FUNCTION_BLOCK "Controle_Dosagem_Complementos"   // FB7, FBD
{ S7_Optimized_Access := 'TRUE' }
VERSION : 0.1
   VAR_INPUT
      inEnable : Bool;
      inBotao_Externo : Bool;
      inValor_Atual_Balanca : Real;
   END_VAR
   VAR_OUTPUT
      outLedBotao_Externo : Bool;
   END_VAR
   VAR_IN_OUT
      Controle : Struct
         Quantidade_Itens : Int;   // Quantidade de complementos na receita
         Item_Atual : Int;   // Em qual item da receita esta no momento
         Quantidade_Dosada_Item_Atual : Real;   // Quantidade dosada do item atual, valor disponível após finalizado dosagem
         Habilitado_Inicio_Dosagem : Bool;   // Habilita o inicio da dosagem manual
         Botao_Inicio_Fim_Dosagem_IHM : Bool;   // Bit para iniciar ou finalizar dosagem pela IHM
         Item_Atual_Iniciado_Dosagem : Bool;   // Se iniciou a dosagem do item atual
         Item_Atual_Finalizado_Dosagem : Bool;   // Se finalizou a dosagem do item atual
         Finalizado_Dosagem_Complementos : Bool;   // Se finalizou a dosagem de todos os complementos
         Reserva : Bool;
         Reserva_1 : Bool;
         Reserva_2 : Bool;
      END_STRUCT;
   END_VAR
   VAR
      Valor_Tara_Balanca : Real;
      Borda_Finalizado_Dosagem_Item : R_TRIG;
   END_VAR
BEGIN

REGION Network 1 (SCL)
   //Maycon Lutz
   //Dosagem de complmento manual na balança

   //O inicio da dosagem pode ser setado por dois lugares, ou por botão fisico, ou na IHM.
   //A finalização da dosagem pode ser setada por dois lugares, ou por botão fisico, ou na IHM.

   //O processo funciona da seguinte maneira, se não esta iniciado a dosagem manual, nem finalizada, é liberado 
   //iniciar uma dosagem em manual, enquanto esta nesse estado, o valor da balança atual é passado para uma variavel
   //como tara da balança, após iniciar a dosagem, paramos de atualizar esse variavel de tara, assim temos um valor 
   //atual de peso da balança antes de iniciar a dosagem manual, após iniciado se apertado no botão novamente
   //é setado o bit de finalizado, e resetado o bit de iniciado, e atualizado a variavel de quantidade dosada,
   //assim sabemos quanto foi dosado manualmente no complementendo especifico. Após o supervisório detectar que 
   //nao esta iniciado e esta finalizado é salvo o valor da dosagem do produto especifico e resetado via supervisório
   //o bit de finalizado, fazendo que habilite a próxima dosagem caso tenha. Assim segue sucessivamente.
   //

   IF #inEnable THEN

       //Somente atualiza o valor da tara e habilita ou não iniciar processo
       IF NOT #Controle.Item_Atual_Iniciado_Dosagem AND NOT #Controle.Item_Atual_Finalizado_Dosagem THEN
           #Valor_Tara_Balanca := #inValor_Atual_Balanca;
           #Controle.Habilitado_Inicio_Dosagem := true;
       ELSE
           #Controle.Habilitado_Inicio_Dosagem := false;

       END_IF;

       //Controle de inicio ou fim atualizados por botão fisico ou por bit da IHM.
       //Verifica se recebeu um pulso do botao externo ou true do bit da ihm
       IF (#inBotao_Externo OR #Controle.Botao_Inicio_Fim_Dosagem_IHM) THEN

           //Verifica se a dosagem esta iniciada, se esta iniciada finaliza
           IF #Controle.Item_Atual_Iniciado_Dosagem THEN
               #Controle.Item_Atual_Finalizado_Dosagem := true;
           ELSE
               //Verifica se esta habilitado a iniciar o processo, se sim set true em iniciar dosagem.
               IF #Controle.Habilitado_Inicio_Dosagem THEN
                   #Controle.Item_Atual_Iniciado_Dosagem := true;
               END_IF;

           END_IF;

           //Reseta bit da IHM.
           IF #Controle.Botao_Inicio_Fim_Dosagem_IHM THEN
               #Controle.Botao_Inicio_Fim_Dosagem_IHM := false;
           END_IF;





       END_IF;

       //Se finalizou a dosagem é resetado o bit de inicio da dosagem e atualizado o valor que foi dosado no item atual.
       IF #Controle.Item_Atual_Finalizado_Dosagem THEN

           #Controle.Item_Atual_Iniciado_Dosagem := false;
           #Controle.Quantidade_Dosada_Item_Atual := #inValor_Atual_Balanca - #Valor_Tara_Balanca;


       END_IF;

       #Borda_Finalizado_Dosagem_Item(CLK := #Controle.Item_Atual_Finalizado_Dosagem);

       IF #Borda_Finalizado_Dosagem_Item.Q THEN
           #Controle.Item_Atual := #Controle.Item_Atual + 1;
       END_IF;


       //Controle do led do botão externo
       IF NOT #Controle.Item_Atual_Iniciado_Dosagem AND NOT #Controle.Item_Atual_Finalizado_Dosagem THEN
           #outLedBotao_Externo := "Clock_1Hz";
       ELSIF #Controle.Item_Atual_Iniciado_Dosagem THEN
           #outLedBotao_Externo := "Clock_2Hz";
           #Controle.Quantidade_Dosada_Item_Atual := #inValor_Atual_Balanca - #Valor_Tara_Balanca;
       ELSE
           #outLedBotao_Externo := false;
       END_IF;


       IF #Controle.Item_Atual >= #Controle.Quantidade_Itens AND NOT #Controle.Item_Atual_Finalizado_Dosagem THEN
           #Controle.Finalizado_Dosagem_Complementos := true;
       END_IF;
   ELSE
       #Controle.Item_Atual := 0;
       #Controle.Item_Atual_Iniciado_Dosagem := false;
       #outLedBotao_Externo := false;
       #Controle.Finalizado_Dosagem_Complementos := false;
       #Controle.Habilitado_Inicio_Dosagem := false;
   END_IF;
END_REGION
END_FUNCTION_BLOCK

FUNCTION_BLOCK "Controle_Automatico_Bateladas"   // FB9, FBD
{ S7_Optimized_Access := 'TRUE' }
VERSION : 0.1
   VAR_IN_OUT
      inOutReceita : Struct
         Peso_Producao_Total : Real;   // Peso da produção total
         Peso_Total_Por_Batelada : Real;   // Peso por batelada
         Peso_Materia_Prima_1 : Real;   // Peso da materia prima 1
         Peso_Materia_Prima_2 : Real;   // peso da materia prima 2
         Silo_Materia_Prima_1 : Int;   // Qual silo esta a materia prima 1
         Silo_Materia_Prima_2 : Int;   // Qual silo esta a materia prima 2
         Quantidade_Bateladas : Int;   // quantidade de bateladas para realizar a produção total
         Quantidade_Complemento_Pre : Int;   // quantidade de complementos pre
         Quantidade_Complemento_Pos : Int;   // quantidade de complementos pos
         Tempo_Mistura_Pre : DInt;   // Tempo de pré mistura
         Tempo_Mistura_Pos : DInt;   // Tempo de pós mistura
      END_STRUCT;
      inOutComando : Struct
         Habilitado_Produzir : Bool;   // Habilita Inicar uma produção
         Ligar_Producao : Bool;   // Liga a produção da receita selecionada
         Em_Producao : Bool;   // Em produção
      END_STRUCT;
   END_VAR
BEGIN
END_FUNCTION_BLOCK

FUNCTION_BLOCK "Controle_Producao_Automatica"   // FB11, FBD
{ S7_Optimized_Access := 'TRUE' }
VERSION : 0.1
BEGIN
END_FUNCTION_BLOCK

// folder: FB/Equipamentos

FUNCTION_BLOCK "PD"   // FB1, FBD
{ S7_Optimized_Access := 'TRUE' }
VERSION : 0.1
   VAR_INPUT
      inConfirmacaoContator : Bool;
      inConfirmcaoDisjuntor : Bool;
      inEmergencia : Bool;
      inLibera : Bool;
      inLigaAutomatico : Bool;
      inTempoFalha : Time;
   END_VAR
   VAR_OUTPUT
      Output_Liga_Bool : Bool;
   END_VAR
   VAR_IN_OUT
      InOutCommand_Control : "typePD";
   END_VAR
   VAR
      Stat_AuxOutputLiga_Bool : Bool;
      Stat_AuxDesligando_Bool : Bool;
      Stat_FalhaConfirmacao_TONTIME : TON_TIME;
      Stat_FalhaDisjuntorNaoDesligou_TONTIME : TON_TIME;
      Stat_NegDisjuntor_Bool : Bool;
      Stat_NegDesligando_Bool : Bool;
      Stat_PosDesligando_Bool : Bool;
      Static_Horimetro : "Horimetro_REV01";
      Stat_NegContator_Bool : Bool;
      Stat_TOF_Desligamento : TOF_TIME;
      Stat_Liberado_Motor : Bool;
      Tempo_Limpeza : DInt;
   END_VAR
   VAR_TEMP   // added for the SCL form of the ladder/FBD networks
      _w1 : Bool;
      _w2 : Bool;
   END_VAR
BEGIN

REGION Network 1 (SCL): Reseta Liga Manual
   // Reseta Liga Manual
   IF #InOutCommand_Control.automatico OR
       (NOT #inLibera AND NOT #InOutCommand_Control.Libera_Bloqueio_Manual) OR
       #InOutCommand_Control.manutencao OR
       NOT #inConfirmcaoDisjuntor OR
       #InOutCommand_Control.falhaGeral OR
       NOT #inEmergencia
   THEN
       #InOutCommand_Control.ligaManual := false;
   END_IF;
END_REGION

REGION Network 2 (SCL): Controle modo Manual/Auto
   //Controle modos 
   IF NOT #InOutCommand_Control.manual AND NOT #InOutCommand_Control.automatico THEN
       #InOutCommand_Control.manual := true;
       //#InOutControl.Automatico := false;
   END_IF;

   IF #InOutCommand_Control.manual AND #InOutCommand_Control.automatico THEN
       #InOutCommand_Control.manual := true;
       //#InOutControl.Automatico := false;

   END_IF;
END_REGION

REGION Network 3: Controle Liga Partida Manual/Automático
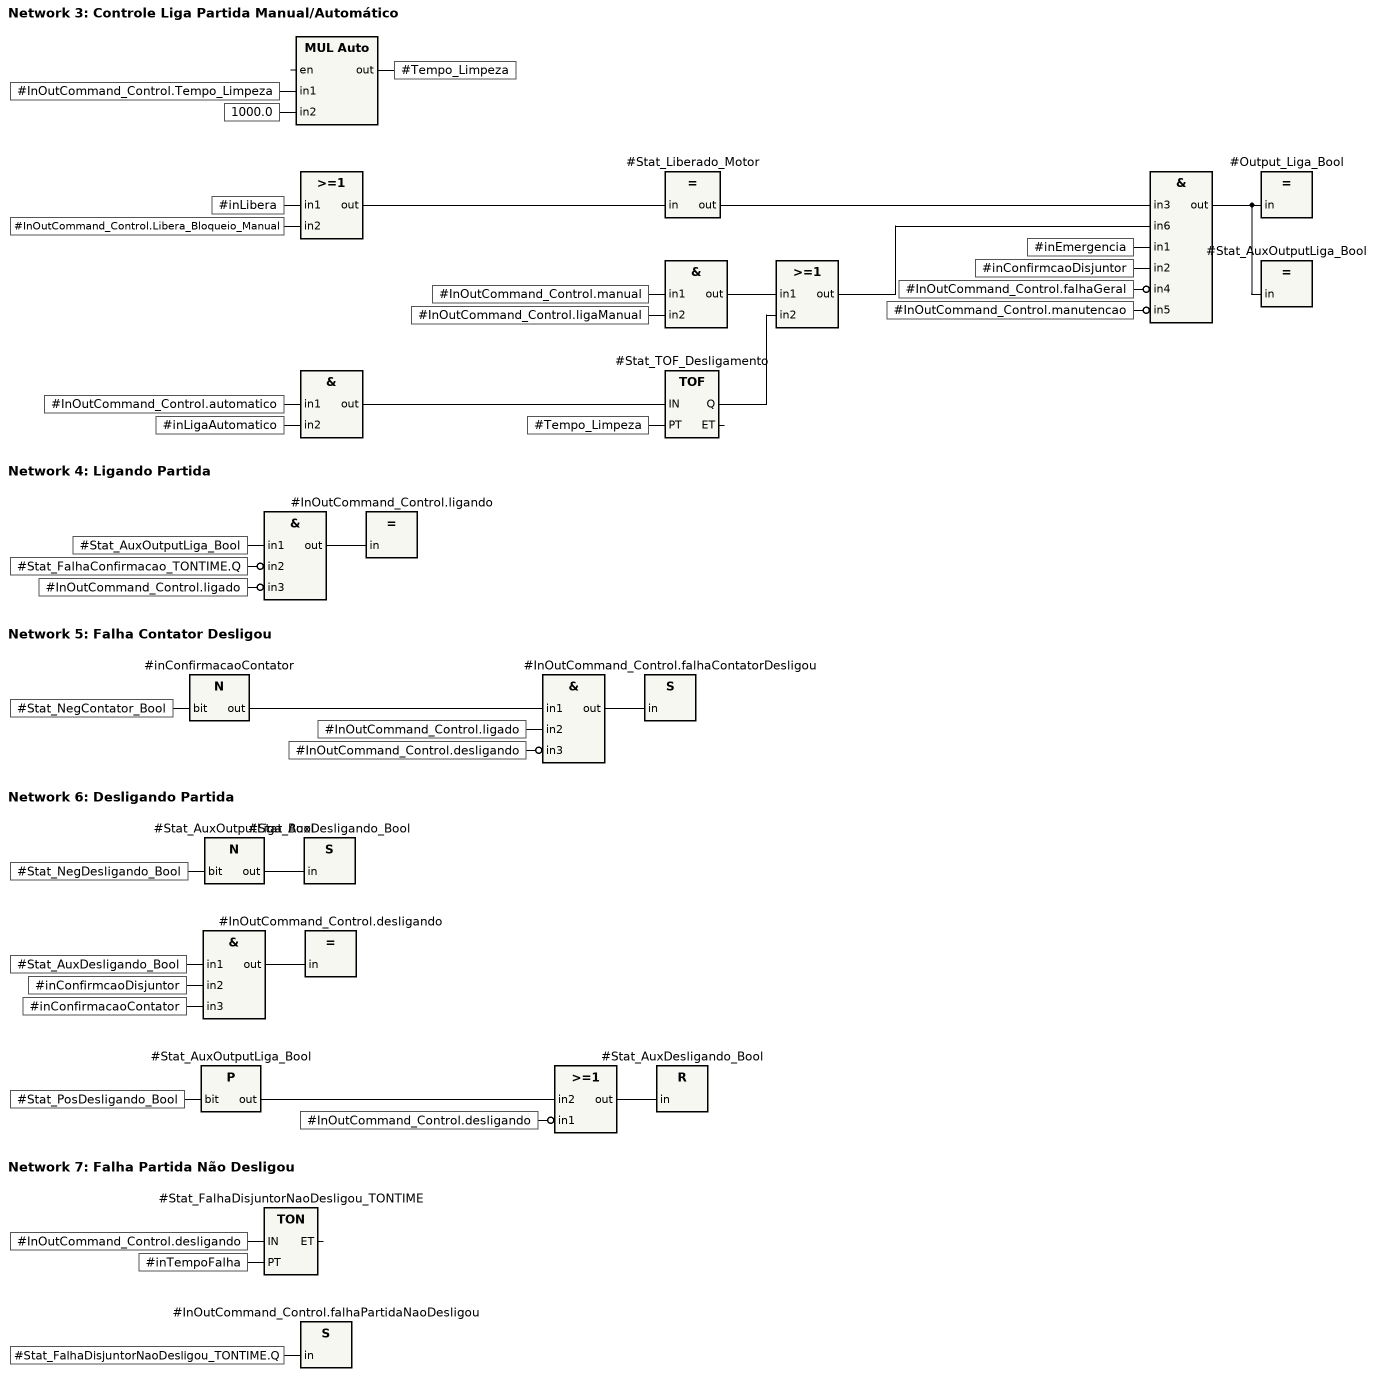
   #Tempo_Limpeza := #InOutCommand_Control.Tempo_Limpeza * 1000.0;
   #Stat_Liberado_Motor := #inLibera OR #InOutCommand_Control.Libera_Bloqueio_Manual;
   #Stat_TOF_Desligamento(IN := #InOutCommand_Control.automatico AND #inLigaAutomatico, PT := #Tempo_Limpeza);   // TOF
   #Output_Liga_Bool := #Stat_Liberado_Motor AND ((#InOutCommand_Control.manual AND #InOutCommand_Control.ligaManual) OR #Stat_TOF_Desligamento.Q) AND #inEmergencia AND #inConfirmcaoDisjuntor AND NOT #InOutCommand_Control.falhaGeral AND NOT #InOutCommand_Control.manutencao;
   #Stat_AuxOutputLiga_Bool := #Output_Liga_Bool;
END_REGION

REGION Network 4: Ligando Partida
   #InOutCommand_Control.ligando := #Stat_AuxOutputLiga_Bool AND NOT #Stat_FalhaConfirmacao_TONTIME.Q AND NOT #InOutCommand_Control.ligado;
END_REGION

REGION Network 5: Falha Contator Desligou
   #_w1 := NOT #inConfirmacaoContator AND #Stat_NegContator_Bool;   // falling edge of #inConfirmacaoContator
   #Stat_NegContator_Bool := #inConfirmacaoContator;
   IF #_w1 AND #InOutCommand_Control.ligado AND NOT #InOutCommand_Control.desligando THEN
       #InOutCommand_Control.falhaContatorDesligou := TRUE;
   END_IF;
END_REGION

REGION Network 6: Desligando Partida
   #_w1 := NOT #Stat_AuxOutputLiga_Bool AND #Stat_NegDesligando_Bool;   // falling edge of #Stat_AuxOutputLiga_Bool
   #Stat_NegDesligando_Bool := #Stat_AuxOutputLiga_Bool;
   IF #_w1 THEN #Stat_AuxDesligando_Bool := TRUE; END_IF;
   #InOutCommand_Control.desligando := #Stat_AuxDesligando_Bool AND #inConfirmcaoDisjuntor AND #inConfirmacaoContator;
   #_w2 := #Stat_AuxOutputLiga_Bool AND NOT #Stat_PosDesligando_Bool;   // rising edge of #Stat_AuxOutputLiga_Bool
   #Stat_PosDesligando_Bool := #Stat_AuxOutputLiga_Bool;
   IF #_w2 OR NOT #InOutCommand_Control.desligando THEN #Stat_AuxDesligando_Bool := FALSE; END_IF;
END_REGION

REGION Network 7: Falha Partida Não Desligou
   #Stat_FalhaDisjuntorNaoDesligou_TONTIME(IN := #InOutCommand_Control.desligando, PT := #inTempoFalha);   // TON
   IF #Stat_FalhaDisjuntorNaoDesligou_TONTIME.Q THEN
       #InOutCommand_Control.falhaPartidaNaoDesligou := TRUE;
   END_IF;
END_REGION

REGION Network 8: Falha Disjuntor Desligou
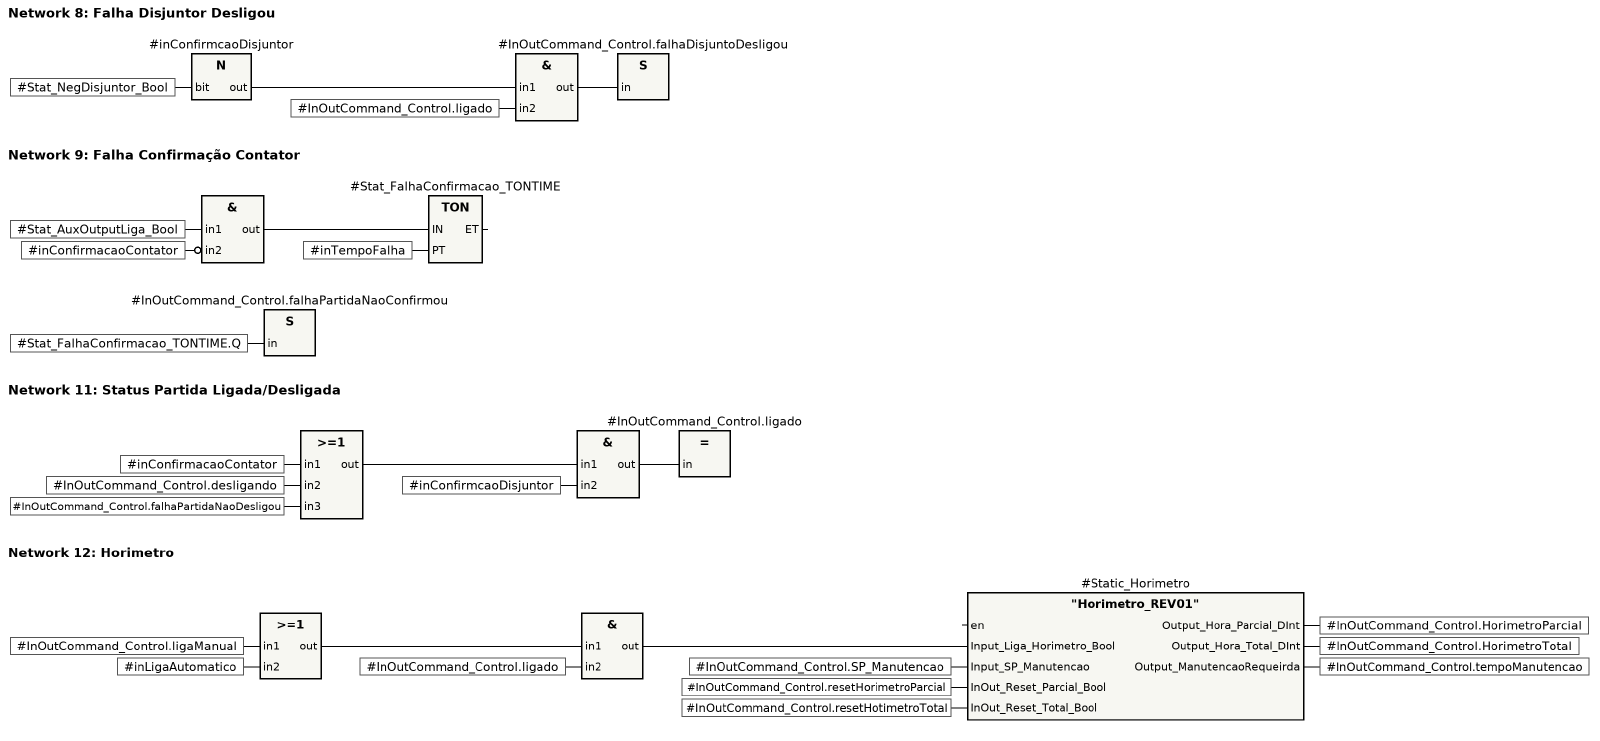
   #_w1 := NOT #inConfirmcaoDisjuntor AND #Stat_NegDisjuntor_Bool;   // falling edge of #inConfirmcaoDisjuntor
   #Stat_NegDisjuntor_Bool := #inConfirmcaoDisjuntor;
   IF #_w1 AND #InOutCommand_Control.ligado THEN #InOutCommand_Control.falhaDisjuntoDesligou := TRUE; END_IF;
END_REGION

REGION Network 9: Falha Confirmação Contator
   // Gera Falha Partida não confirmou
   #Stat_FalhaConfirmacao_TONTIME(IN := #Stat_AuxOutputLiga_Bool AND NOT #inConfirmacaoContator,   // TON
                           PT := #inTempoFalha);
   IF #Stat_FalhaConfirmacao_TONTIME.Q THEN #InOutCommand_Control.falhaPartidaNaoConfirmou := TRUE; END_IF;
END_REGION

REGION Network 10 (SCL): Falha Geral
       //Falha Geral
       IF #InOutCommand_Control.falhaPartidaNaoConfirmou OR
           #InOutCommand_Control.falhaContatorDesligou OR
           #InOutCommand_Control.falhaDisjuntoDesligou OR
           #InOutCommand_Control.falhaPartidaNaoDesligou
       THEN
           #InOutCommand_Control.falhaGeral := true;
       ELSE
           #InOutCommand_Control.falhaGeral := false;
       END_IF;
END_REGION

REGION Network 11: Status Partida Ligada/Desligada
   #InOutCommand_Control.ligado := (#inConfirmacaoContator OR #InOutCommand_Control.desligando OR #InOutCommand_Control.falhaPartidaNaoDesligou) AND #inConfirmcaoDisjuntor;
END_REGION

REGION Network 12: Horimetro
   #Static_Horimetro(Input_Liga_Horimetro_Bool := (#InOutCommand_Control.ligaManual OR #inLigaAutomatico) AND #InOutCommand_Control.ligado,   // "Horimetro_REV01"
                     Input_SP_Manutencao := #InOutCommand_Control.SP_Manutencao,
                     InOut_Reset_Parcial_Bool := #InOutCommand_Control.resetHorimetroParcial,
                     InOut_Reset_Total_Bool := #InOutCommand_Control.resetHotimetroTotal,
                     Output_Hora_Parcial_DInt => #InOutCommand_Control.HorimetroParcial,
                     Output_Hora_Total_DInt => #InOutCommand_Control.HorimetroTotal,
                     Output_ManutencaoRequeirda => #InOutCommand_Control.tempoManutencao);
END_REGION

REGION Network 13 (SCL): Status Supervisorio
   //Sinais Supervisório
   #InOutCommand_Control.liberado := #Stat_Liberado_Motor;
   #InOutCommand_Control.emergencia := #inEmergencia;
   #InOutCommand_Control.disjuntorDesligado := NOT #inConfirmcaoDisjuntor;
END_REGION

REGION Network 14 (SCL): Reset Falhas
   //Reset Falhas
   IF #InOutCommand_Control.reset THEN

       #InOutCommand_Control.falhaPartidaNaoConfirmou := false;
       #InOutCommand_Control.falhaContatorDesligou := false;
       #InOutCommand_Control.falhaDisjuntoDesligou := false;
       #InOutCommand_Control.falhaPartidaNaoDesligou := false;

       #InOutCommand_Control.reset := false;
   END_IF;
END_REGION
END_FUNCTION_BLOCK

FUNCTION_BLOCK "Atuador_Linear_Digital"   // FB2, FBD
TITLE = Controle atuador com retorno de posição por fim de curso com dois lados (aberto, fechado)
{ S7_Optimized_Access := 'TRUE' }
VERSION : 0.1
// Maycon Lutz
// 15/07/20
// 
// Lado 1 - Considerado Aberto
// Lado 2 - Considerado Fechado
   VAR_INPUT
      inConfirmacao_Contator_Lado1 : Bool;
      inConfirmacao_Contator_Lado2 : Bool;
      inSensor_Lado1 : Bool;
      inSensor_Lado2 : Bool;
      inAciona_Lado1_Auto : Bool;
      inAciona_Lado2_Auto : Bool;
      inTempo_Falha : Time;
      inEmergencia : Bool;
      inLibera : Bool;
   END_VAR
   VAR_OUTPUT
      outAciona_Lado1 : Bool;
      outAciona_Lado2 : Bool;
      outEm_Posicao_Lado1 : Bool;
      outEm_Posicao_Lado2 : Bool;
   END_VAR
   VAR_IN_OUT
      Command : "typeAtuadorLinearDigital";
   END_VAR
   VAR
      Liberado : Bool;
      Intertravamento_Modo_Digital : Bool;
      Temporizador_Intertravamento : TON_TIME;
      Temporizador_Falha_Acionamento : TON_TIME;
      Temporizador_Falha_Contator_Lado1 : TON_TIME;
      Temporizador_Falha_Contator_Lado2 : TON_TIME;
      R_Trig_Manual : R_TRIG;
      R_Trig_Automatico : R_TRIG;
   END_VAR
BEGIN

REGION Network 1 (SCL): Controle modo Manual e Automático
   #R_Trig_Manual(CLK := #Command.Manual);
   //borda de subida em manual, false em automatico
   IF #R_Trig_Manual.Q THEN
       #Command.Automatico := false;
   END_IF;

   //borda de subida em automatico, false em manual
   #R_Trig_Automatico(CLK := #Command.Automatico);

   IF #R_Trig_Automatico.Q THEN
       #Command.Manual := false;
   END_IF;

   //Se os dois bits em true, false em automatico
   IF #Command.Manual AND #Command.Automatico THEN
       #Command.Automatico := false;
   END_IF;

   //se os dois bits em false, true em manual
   IF NOT #Command.Manual AND NOT #Command.Automatico THEN
       #Command.Manual := true;
   END_IF;
END_REGION

REGION Network 2 (SCL): Status Sensores
   #Command.Em_Posicao_Lado1 := #inSensor_Lado1;
   #Command.Em_Posicao_Lado2 := #inSensor_Lado2;
   #outEm_Posicao_Lado1 := #inSensor_Lado1;
   #outEm_Posicao_Lado2 := #inSensor_Lado2;
END_REGION

REGION Network 3 (SCL): Condições Liberação Funcionamento
   IF #inEmergencia AND //emergencia
       (#inLibera OR #Command.Libera_Bloqueio_Manual) AND //liberado
       NOT #Command.Falha_Acionando_Lado1 AND // falha acionamento lado 1
       NOT #Command.Falha_Acionando_Lado2 AND //falha acionamento lado 2
       NOT #Command.Falha_2_Posicoes_Ativa AND
       NOT #Command.Falha_Confirmacao_Contator_Lado1 AND
       NOT #Command.Falha_Confirmacao_Contator_Lado2 AND 
       NOT #Command.Manutencao AND // em manutenção
       NOT (#inAciona_Lado1_Auto AND #inAciona_Lado2_Auto)//acionado 2 lado ao mesmo tempo em auto
   THEN
       #Liberado := true;
   ELSE
       #Liberado := false;

       //Verifica se esta aberto o registro em manual ou em automático e solicita fechar
       IF #Command.Em_Posicao_Lado1 OR NOT #Command.Em_Posicao_Lado2 AND
           (
           #Command.Falha_2_Posicoes_Ativa OR
           #Command.Falha_Acionando_Lado1 OR
           #Command.Falha_Acionando_Lado2 OR
           #Command.Falha_Confirmacao_Contator_Lado1 OR
           #Command.Falha_Confirmacao_Contator_Lado2
           )
       THEN
           #Command.Aciona_Lado2 := true;

       END_IF;
       #Command.Aciona_Lado1 := false;
   END_IF;
END_REGION

REGION Network 4 (SCL): Status das condições
   #Command.Em_Emergencia := #inEmergencia;
   #Command.Liberado := #Liberado;
END_REGION

REGION Network 5 (SCL): Acionamento

   IF #Command.Automatico THEN
       #Command.Aciona_Lado1 := false;
       #Command.Aciona_Lado2 := false;
   END_IF;



   //Verifica se estava acionado de um lado e foi solicitado outro lado
   //assim reseta o lado anterior e intertrava o lado novo solicitado
   //evitando problemas em campo.
   IF #Command.Aciona_Lado1 AND
       #Command.Aciona_Lado2 THEN

       #Intertravamento_Modo_Digital := true;

       IF #Command.Acionando_Lado1 THEN

           #Command.Aciona_Lado1 := false;
       END_IF;

       IF #Command.Acionando_Lado2 THEN

           #Command.Aciona_Lado2 := false;
       END_IF;

   END_IF;


   //temporizador de intertravamento quando solicitado dois lados ao mesmo tempo
   #Temporizador_Intertravamento(IN := #Intertravamento_Modo_Digital, PT := T#3S);

   //libera intertravamento
   IF #Temporizador_Intertravamento.Q THEN
       #Intertravamento_Modo_Digital := false;
   END_IF;


   //acionamento lado 1
   IF ((#Command.Aciona_Lado1 AND
       NOT #Intertravamento_Modo_Digital AND
       #Command.Manual) OR
       (#inAciona_Lado1_Auto AND
       #Command.Automatico
       ))
       AND #Liberado
   THEN

       //quando chegou na posição para de acionar e reseta o aciona lado
       IF #Command.Em_Posicao_Lado1 THEN
           #Command.Aciona_Lado1 := false;
           #Command.Acionando_Lado1 := false;
           #outAciona_Lado1 := false;

       ELSE
           //aciona lado 1
           #Command.Acionando_Lado1 := true;
           #outAciona_Lado1 := true;
       END_IF;
   ELSE

       #Command.Acionando_Lado1 := false;
       #outAciona_Lado1 := false;

   END_IF;

   //acionamento lado 2
   IF ((#Command.Aciona_Lado2 AND
       NOT #Intertravamento_Modo_Digital AND
       #Command.Manual) OR
       (#inAciona_Lado2_Auto AND
       #Command.Automatico
       ))
   //Não verifica se esta liberado ou não pois para fechar o registro não precisar estar liberado, somente para abrir.
   THEN

       //quando chegou na posição para de acionar e reseta o aciona lado
       IF #Command.Em_Posicao_Lado2 THEN
           #Command.Aciona_Lado2 := false;
           #Command.Acionando_Lado2 := false;
           #outAciona_Lado2 := false;
       ELSE
           //aciona lado 2
           #Command.Acionando_Lado2 := true;
           #outAciona_Lado2 := true;
       END_IF;
   ELSE

       #Command.Acionando_Lado2 := false;
       #outAciona_Lado2 := false;

   END_IF;
END_REGION

REGION Network 6 (SCL): Falha confirmação contatores

   #Temporizador_Falha_Contator_Lado1(IN := #outAciona_Lado1 AND NOT #inConfirmacao_Contator_Lado1,
                                      PT := t#3s);

   #Temporizador_Falha_Contator_Lado2(IN := #outAciona_Lado2 AND NOT #inConfirmacao_Contator_Lado2,
                                      PT := t#3s);

   IF #Temporizador_Falha_Contator_Lado1.Q THEN
       #Command.Falha_Confirmacao_Contator_Lado1 := true;
   END_IF;

   IF #Temporizador_Falha_Contator_Lado2.Q THEN
       #Command.Falha_Confirmacao_Contator_Lado2 := true;
   END_IF;
END_REGION

REGION Network 7 (SCL): Falha 2 posições ativas
   IF #Command.Em_Posicao_Lado1 AND #Command.Em_Posicao_Lado2 THEN
       #Command.Falha_2_Posicoes_Ativa := true;
   END_IF;
END_REGION

REGION Network 8 (SCL): Falha acionamento - Sensor não encontrado
   //conta tempo para falha de acionamento
   #Temporizador_Falha_Acionamento(IN := (#Command.Acionando_Lado1 OR #Command.Acionando_Lado2),
                                   PT := #inTempo_Falha);
   //falha de acionamento
   IF #Temporizador_Falha_Acionamento.Q THEN
       IF #Command.Acionando_Lado1 THEN
           #Command.Falha_Acionando_Lado1 := true;
       END_IF;

       IF #Command.Acionando_Lado2 THEN
           #Command.Falha_Acionando_Lado2 := true;
       END_IF;

   END_IF;
END_REGION

REGION Network 9 (SCL): Reset Falha
   //reset falha de acionamento
   IF #Command.Reset_Falha THEN
       #Command.Falha_Acionando_Lado1 := false;
       #Command.Falha_Acionando_Lado2 := false;
       #Command.Falha_2_Posicoes_Ativa := false;
       #Command.Falha_Confirmacao_Contator_Lado1 := false;
       #Command.Falha_Confirmacao_Contator_Lado2 := false;
       #Command.Reset_Falha := false;
   END_IF;
END_REGION
END_FUNCTION_BLOCK

FUNCTION_BLOCK "Atuador_Linear_Analogico"   // FB3, LAD
TITLE = Controle atuador com retorno de posição analógico 0-100% ou fim de curso com dois lados (aberto, fechado)
{ S7_Optimized_Access := 'TRUE' }
VERSION : 0.1
// Maycon Lutz
// 15/07/20
// 
// relacionamos modo analógico quando temos retorno de posição do atuador de 0 - 100%
// relacionamos modo digital quando temos retorno de posição com fim de curso um em cada lado.
// AMBOS SÃO ACIONADOS DIGITALMENTE PARA UM LADO OU PARA OUTRO LADO.
   VAR_INPUT
      inConfirmacao_Contator_Lado1 : Bool;
      inConfirmacao_Contator_Lado2 : Bool;
      inFalha_Leitura_Posicao : Bool;
      inTolerancia_Erro_Posicao : Real;   // Tolerancia de erro entre a posicação solicitada e a posição atual - valor de 0 - 100%
      inPosicao_Atual : Real;   // Posicao atual - valor de 0 - 100%
      inPosicao_Solicitada_Automatico : Real;
      inTempo_Falha : Time;
      inEmergencia : Bool;
      inLibera : Bool;
      inLiga_Automatico : Bool;
   END_VAR
   VAR_OUTPUT
      outAciona_Lado1 : Bool;
      outAciona_Lado2 : Bool;
      outPosicao_Atual : Bool;
   END_VAR
   VAR_IN_OUT
      Command : "typeAtuadorLinearAnalogico";
   END_VAR
   VAR
      Liberado : Bool;
      Intertravamento : Bool;
      Posicionar : Bool;
      Solicita_Posicionar : Bool;
      Posicao_Posicionar : Real;
      Temporizador_Falha_Leitura_Posicao : TON_TIME;
      Temporizador_Falha_Posicionamento : TON_TIME;
      Temporizador_Libera_Acionamento : TON_TIME;
      Temporizador_Falha_Contator_Lado1 : TON_TIME;
      Temporizador_Falha_Contator_Lado2 : TON_TIME;
      R_Trig_Manual : R_TRIG;
      R_Trig_Automatico : R_TRIG;
      Posicao_Solicitada_Manual_OLD : Real;
   END_VAR
BEGIN

REGION Network 1 (SCL): Controle modo Manual e Automático
   #R_Trig_Manual(CLK := #Command.Manual);
   //borda de subida em manual, false em automatico
   IF #R_Trig_Manual.Q THEN
       #Command.Automatico := false;
   END_IF;

   //borda de subida em automatico, false em manual
   #R_Trig_Automatico(CLK := #Command.Automatico);

   IF #R_Trig_Automatico.Q THEN
       #Command.Manual := false;
   END_IF;

   //Se os dois bits em true, false em automatico
   IF #Command.Manual AND #Command.Automatico THEN
       #Command.Automatico := false;
   END_IF;

   //se os dois bits em false, true em manual
   IF NOT #Command.Manual AND NOT #Command.Automatico THEN
       #Command.Manual := true;
   END_IF;
END_REGION

REGION Network 2 (SCL): Condições Liberação Funcionamento
   IF #inEmergencia AND //emergencia
       (#inLibera OR #Command.Libera_Bloqueio_Manual) AND //liberado
       NOT #Command.Falha_Leitura_Posicao AND
       NOT #Command.Falha_Posicionamento AND 
       NOT #Command.Falha_Confirmacao_Contator_Lado1 AND
       NOT #Command.Falha_Confirmacao_Contator_Lado2 AND 
       NOT #Command.Manutencao // em manutenção
   THEN
       #Liberado := true;
   ELSE
       #Liberado := false;
   END_IF;
END_REGION

REGION Network 3 (SCL): Status das condições
   #Command.Em_Emergencia := #inEmergencia;
   #Command.Liberado := #inLibera;
END_REGION

REGION Network 4 (SCL): Atualiza valores na palavra de comando
   #Command.Posicao_Atual := #inPosicao_Atual;
   #Command.Posicao_Solicitada_Automatico := #inPosicao_Solicitada_Automatico;
END_REGION

REGION Network 5 (SCL): Posicao Solicitada / posição atual e controle de erro de posicao
END_REGION

REGION Network 6 (SCL): Acionamento Manual

   //Temporizador para liberar alterar a posição novamente após tempo definido
   #Temporizador_Libera_Acionamento(IN := NOT #outAciona_Lado1 AND NOT #outAciona_Lado2,
                                    PT := t#2s);

   //Solicita alteração na posição
   IF (#Command.SP_Posicao_Manual <> #Posicao_Solicitada_Manual_OLD AND
       #Temporizador_Libera_Acionamento.Q AND
       #Liberado AND
       #Command.Manual AND
       #Command.Liga_Manual)
   THEN
       #Posicao_Solicitada_Manual_OLD := #Command.SP_Posicao_Manual;
       #Posicionar := true;
   END_IF;

   //Solicita posicionar
   IF #Posicionar THEN

       //Verifica o lado que necessita atuar
       IF #Command.Posicao_Atual > #Command.SP_Posicao_Manual AND NOT #Solicita_Posicionar THEN
           //Solicita fechar atuador
           #outAciona_Lado1 := true;
           #Solicita_Posicionar := true;
           #Posicao_Posicionar := #Command.SP_Posicao_Manual;
       ELSIF #Command.Posicao_Atual < #Command.SP_Posicao_Manual AND NOT #Solicita_Posicionar THEN
           //Solicita abrir atuador
           #outAciona_Lado2 := true;
           #Solicita_Posicionar := true;
           #Posicao_Posicionar := #Command.SP_Posicao_Manual;
       END_IF;

       //Verifica a posição atual e a posição solicitada e define se chegou a posição correta
       IF #outAciona_Lado2 AND
          #Command.Posicao_Atual >= #Posicao_Posicionar THEN
          #Posicionar := false;
       END_IF;

       IF #outAciona_Lado1 AND
           #Command.Posicao_Atual <= #Posicao_Posicionar THEN
           #Posicionar := false;
       END_IF;

   ELSE
       #outAciona_Lado1 := false;
       #outAciona_Lado2 := false;
       #Solicita_Posicionar := false;
       #Posicao_Posicionar := 0;
   END_IF;
END_REGION

REGION Network 7 (SCL): Atualiza palavra de controle Ligando lado 1/ Ligando lado 2
   #Command.Aciona_Lado1 := #outAciona_Lado1;
   #Command.Aciona_Lado2 := #outAciona_Lado2;
END_REGION

REGION Network 8 (SCL): Falha Confirmação Contatores

   #Temporizador_Falha_Contator_Lado1(IN := #outAciona_Lado1 AND NOT #inConfirmacao_Contator_Lado1,
                                      PT := t#3s);

   #Temporizador_Falha_Contator_Lado2(IN := #outAciona_Lado2 AND NOT #inConfirmacao_Contator_Lado2,
                                      PT := t#3s);

   IF #Temporizador_Falha_Contator_Lado1.Q THEN
       #Command.Falha_Confirmacao_Contator_Lado1 := true;
   END_IF;

   IF #Temporizador_Falha_Contator_Lado2.Q THEN
       #Command.Falha_Confirmacao_Contator_Lado2 := true;
   END_IF;
END_REGION

REGION Network 9 (SCL): Falha Posicionamento
   #Temporizador_Falha_Posicionamento(IN := #Posicionar AND (#Command.Liga_Manual OR #inLiga_Automatico),
                                      PT := #inTempo_Falha);

   IF #Temporizador_Falha_Posicionamento.Q THEN
       #Command.Falha_Posicionamento := true;
   END_IF;
END_REGION

REGION Network 10 (SCL): Falha Leitura Posição
   #Temporizador_Falha_Leitura_Posicao(IN := #inFalha_Leitura_Posicao,
                                       PT := t#3s);

   IF #Temporizador_Falha_Leitura_Posicao.Q THEN
       #Command.Falha_Leitura_Posicao := true;
   END_IF;
END_REGION

REGION Network 11 (SCL): Reset Falha
   //reset falha de acionamento
   IF #Command.Reset_Falha THEN
       #Command.Falha_Leitura_Posicao := false;
       #Command.Falha_Posicionamento := false;
       #Command.Falha_Confirmacao_Contator_Lado1 := false;
       #Command.Falha_Confirmacao_Contator_Lado2 := false;
       #Command.Reset_Falha := false;
   END_IF;
END_REGION
END_FUNCTION_BLOCK

FUNCTION_BLOCK "SS_MOINHO"   // FB4, FBD
{ S7_Optimized_Access := 'TRUE' }
VERSION : 0.1
   VAR_INPUT
      inConfirmacaoContator_Sentido1 : Bool;
      inConfirmacaoContator_Sentido2 : Bool;
      inConfirmcaoDisjuntor : Bool;
      inEmergencia : Bool;
      inLibera : Bool;
      inLigaAutomatico : Bool;
      inTempoFalha : Time;
      inCorrente_Atual : Real;
      inFalha_Leitura_Corrente : Bool;
      inSimulacao : Bool;
   END_VAR
   VAR_OUTPUT
      outLigaSentido1 : Bool;
      outLigaSentido2 : Bool;
      outLigaSoftStarter : Bool;
   END_VAR
   VAR_IN_OUT
      InOutCommand_Control : "typeSS";
   END_VAR
   VAR
      Stat_AuxOutputLiga_Bool : Bool;
      Stat_AuxDesligando_Bool : Bool;
      Stat_FalhaConfirmacao_TONTIME : TON_TIME;
      Stat_FalhaDisjuntorNaoDesligou_TONTIME : TON_TIME;
      Stat_NegDisjuntor_Bool : Bool;
      Stat_NegDesligando_Bool : Bool;
      Stat_PosDesligando_Bool : Bool;
      Static_Horimetro : "Horimetro_REV01";
      Static_Aux_Falha_Geral_Bool : Bool;
      Stat_NegContator_Bool : Bool;
      Stat_NegContator2_Bool : Bool;
      Stat_TOF_Desligamento : TOF_TIME;
      Stat_Liberado_Motor : Bool;
      Tempo_Limpeza : DInt;
   END_VAR
   VAR RETAIN
      Sentido_Giro : Bool;
   END_VAR
   VAR
      Libera_Inverter_Sentido_Giro : TON_TIME;
   END_VAR
   VAR RETAIN
      Tempo_Sentido_Giro : TONR_TIME;
   END_VAR
   VAR
      SP_Tempo_Sentido_Giro : DInt;
      Timer_Desliga_Contatores : TOF_TIME;
      Timer_Liga_SoftStarter : TON_TIME;
   END_VAR
   VAR_TEMP   // added for the SCL form of the ladder/FBD networks
      _w1 : Bool;
      _w2 : Bool;
   END_VAR
BEGIN

REGION Network 1 (SCL): Reseta Liga Manual
   // Reseta Liga Manual
   IF #InOutCommand_Control.automatico OR
       (NOT #inLibera AND NOT #InOutCommand_Control.Libera_Bloqueio_Manual) OR
       #InOutCommand_Control.manutencao OR
       NOT #inConfirmcaoDisjuntor OR
       #Static_Aux_Falha_Geral_Bool
   THEN
       #InOutCommand_Control.ligaManual := false;
   END_IF;
END_REGION

REGION Network 2 (SCL): Controle modo Manual/Auto
   //Controle modos 
   IF NOT #InOutCommand_Control.manual AND NOT #InOutCommand_Control.automatico THEN
       #InOutCommand_Control.manual := true;
       //#InOutControl.Automatico := false;
   END_IF;

   IF #InOutCommand_Control.manual AND #InOutCommand_Control.automatico THEN
       #InOutCommand_Control.manual := true;
       //#InOutControl.Automatico := false;

   END_IF;
END_REGION

REGION Network 3 (SCL): Corrente Atual
   IF NOT #inSimulacao THEN
       #InOutCommand_Control.Corrente_Atual := #inCorrente_Atual;
   END_IF;
END_REGION

REGION Network 4 (SCL): Controle Sentido de Giro
   #Libera_Inverter_Sentido_Giro(IN := NOT #Stat_AuxOutputLiga_Bool,
                                 PT := t#20s);

   #SP_Tempo_Sentido_Giro := (#InOutCommand_Control.SP_Tempo_Reversao * 1000)*60;

   //Conta tempo motor ligado
   #Tempo_Sentido_Giro(IN := #Stat_AuxOutputLiga_Bool,
                       PT := #SP_Tempo_Sentido_Giro);


   //Habilita troca de sentido de giro
   IF #Libera_Inverter_Sentido_Giro.Q THEN

       IF #InOutCommand_Control.inverterSentidoGiro THEN
           #Sentido_Giro := NOT #Sentido_Giro;
           #InOutCommand_Control.inverterSentidoGiro := false;
           RESET_TIMER(#Tempo_Sentido_Giro);
       END_IF;

       IF #Tempo_Sentido_Giro.ET >= #InOutCommand_Control.SP_Tempo_Reversao THEN
           #Sentido_Giro := NOT #Sentido_Giro;
           RESET_TIMER(#Tempo_Sentido_Giro);
       END_IF;
   ELSE
       #InOutCommand_Control.inverterSentidoGiro := false;

   END_IF;



   //Sentido de giro atual
   #InOutCommand_Control.SentidoGiro := #Sentido_Giro;
   //Tempo atual reversão
   #InOutCommand_Control.Tempo_Reversao_Atual := (#Tempo_Sentido_Giro.ET /1000)/60;
END_REGION

REGION Network 5: Controle Liga Partida Manual/Automático
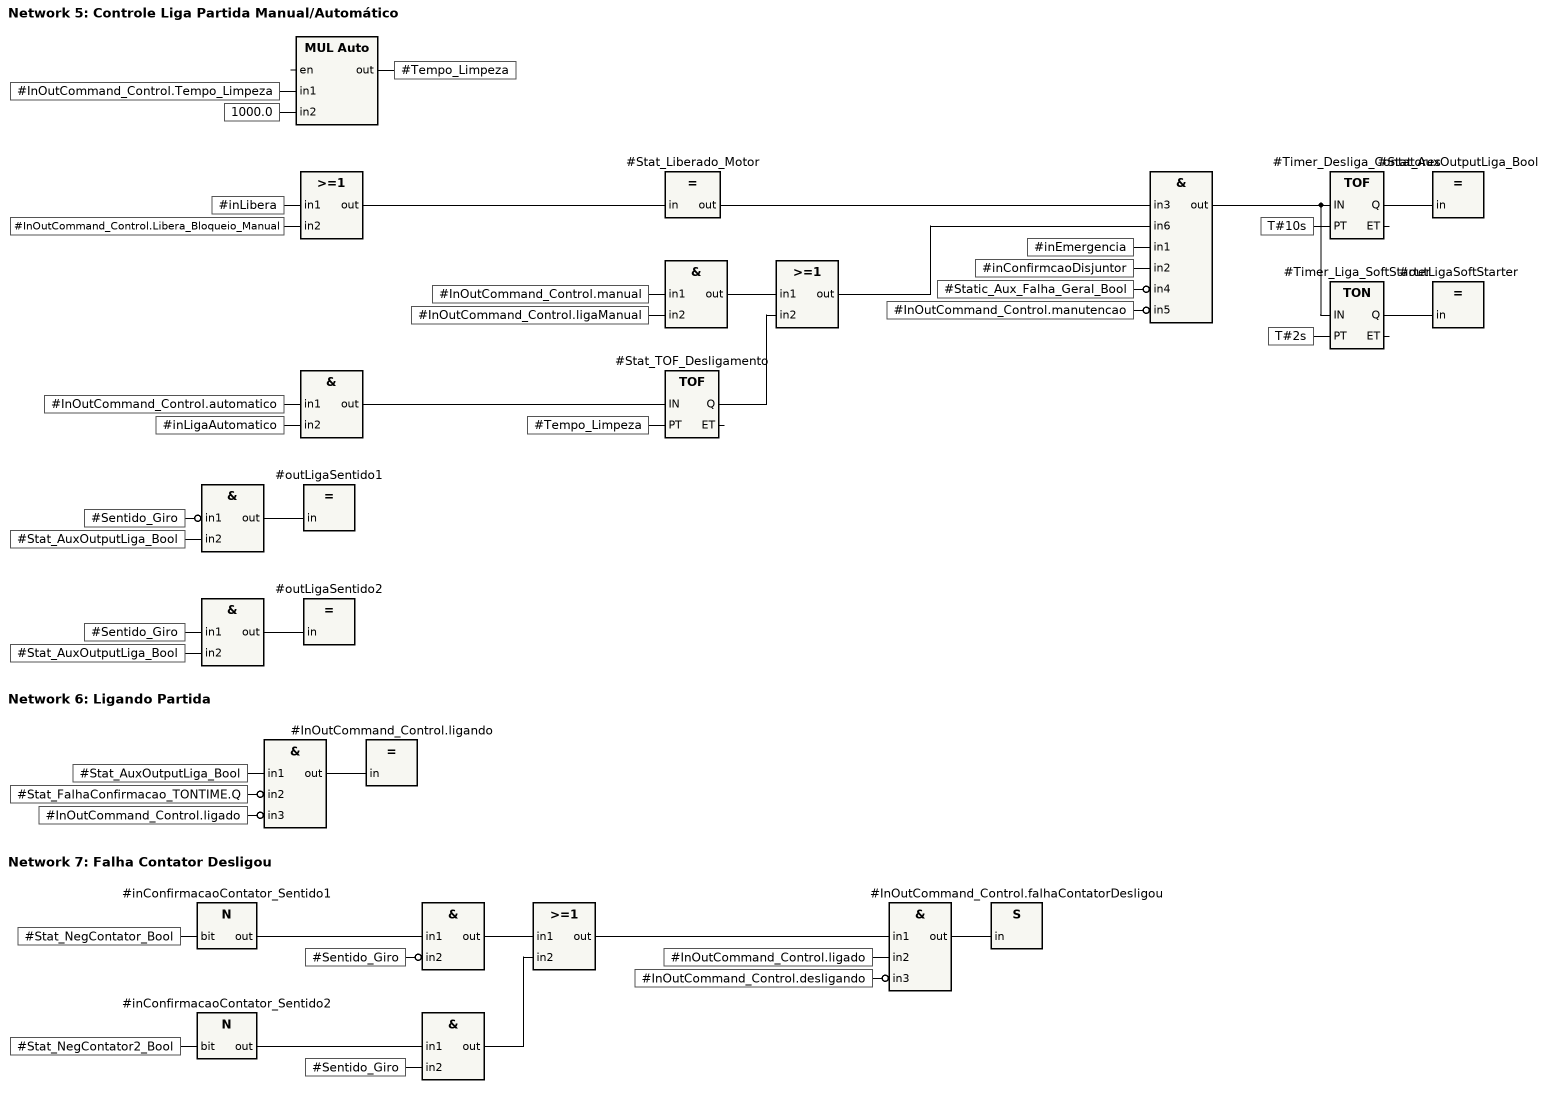
   #Tempo_Limpeza := #InOutCommand_Control.Tempo_Limpeza * 1000.0;
   #Stat_Liberado_Motor := #inLibera OR #InOutCommand_Control.Libera_Bloqueio_Manual;
   #Stat_TOF_Desligamento(IN := #InOutCommand_Control.automatico AND #inLigaAutomatico, PT := #Tempo_Limpeza);   // TOF
   #_w1 := #Stat_Liberado_Motor AND ((#InOutCommand_Control.manual AND #InOutCommand_Control.ligaManual) OR #Stat_TOF_Desligamento.Q) AND #inEmergencia AND #inConfirmcaoDisjuntor AND NOT #Static_Aux_Falha_Geral_Bool AND NOT #InOutCommand_Control.manutencao;
   #Timer_Desliga_Contatores(IN := #_w1, PT := T#10s);   // TOF
   #Stat_AuxOutputLiga_Bool := #Timer_Desliga_Contatores.Q;
   #Timer_Liga_SoftStarter(IN := #_w1, PT := T#2s);   // TON
   #outLigaSoftStarter := #Timer_Liga_SoftStarter.Q;
   #outLigaSentido1 := NOT #Sentido_Giro AND #Stat_AuxOutputLiga_Bool;
   #outLigaSentido2 := #Sentido_Giro AND #Stat_AuxOutputLiga_Bool;
END_REGION

REGION Network 6: Ligando Partida
   #InOutCommand_Control.ligando := #Stat_AuxOutputLiga_Bool AND NOT #Stat_FalhaConfirmacao_TONTIME.Q AND NOT #InOutCommand_Control.ligado;
END_REGION

REGION Network 7: Falha Contator Desligou
   #_w1 := NOT #inConfirmacaoContator_Sentido1 AND #Stat_NegContator_Bool;   // falling edge of #inConfirmacaoContator_Sentido1
   #Stat_NegContator_Bool := #inConfirmacaoContator_Sentido1;
   #_w2 := NOT #inConfirmacaoContator_Sentido2 AND #Stat_NegContator2_Bool;   // falling edge of #inConfirmacaoContator_Sentido2
   #Stat_NegContator2_Bool := #inConfirmacaoContator_Sentido2;
   IF ((#_w1 AND NOT #Sentido_Giro) OR (#_w2 AND #Sentido_Giro)) AND #InOutCommand_Control.ligado AND NOT #InOutCommand_Control.desligando THEN
       #InOutCommand_Control.falhaContatorDesligou := TRUE;
   END_IF;
END_REGION

REGION Network 8: Desligando Partida
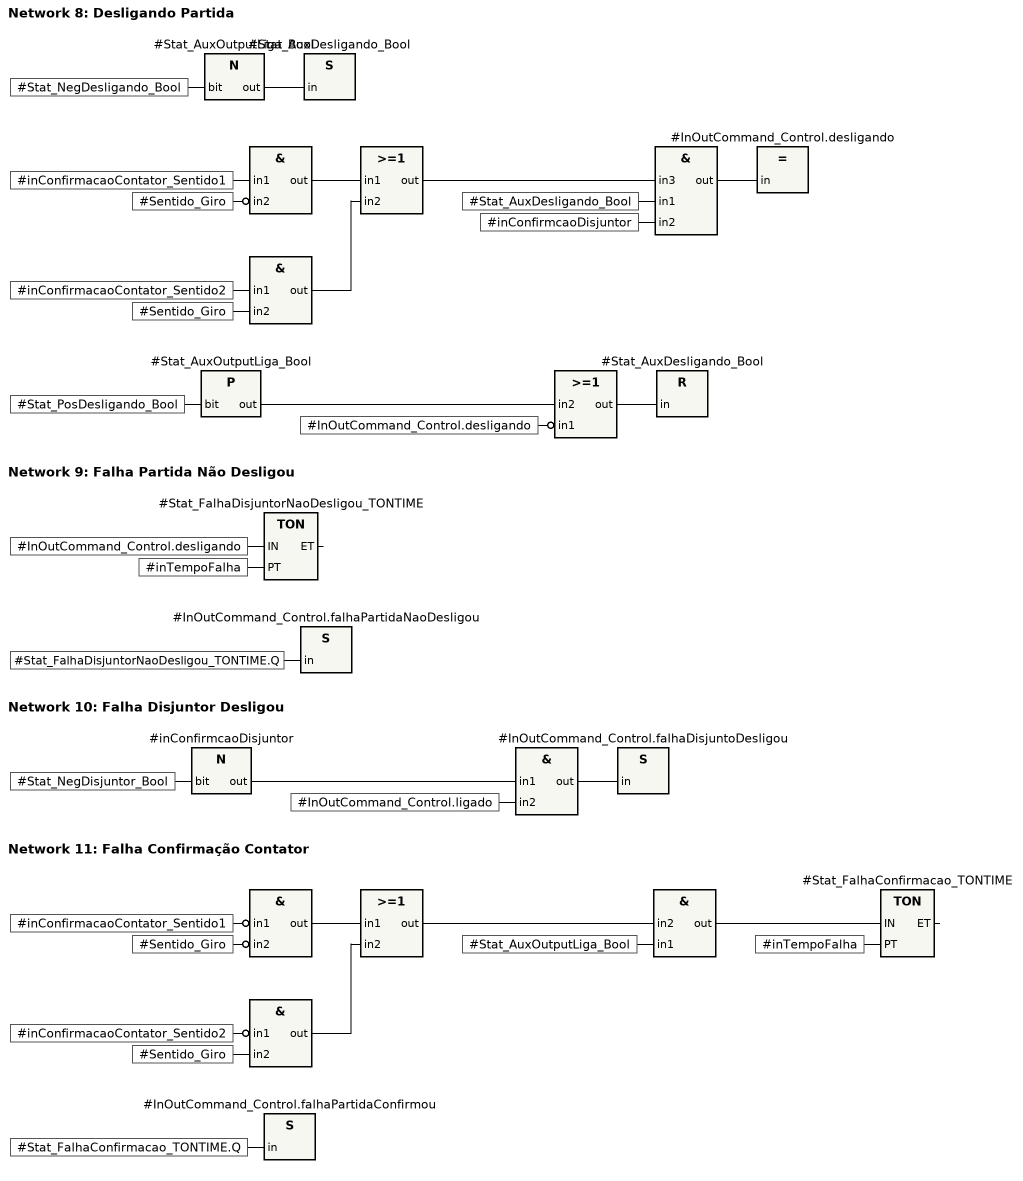
   #_w1 := NOT #Stat_AuxOutputLiga_Bool AND #Stat_NegDesligando_Bool;   // falling edge of #Stat_AuxOutputLiga_Bool
   #Stat_NegDesligando_Bool := #Stat_AuxOutputLiga_Bool;
   IF #_w1 THEN #Stat_AuxDesligando_Bool := TRUE; END_IF;
   #InOutCommand_Control.desligando := ((#inConfirmacaoContator_Sentido1 AND NOT #Sentido_Giro) OR (#inConfirmacaoContator_Sentido2 AND #Sentido_Giro)) AND #Stat_AuxDesligando_Bool AND #inConfirmcaoDisjuntor;
   #_w2 := #Stat_AuxOutputLiga_Bool AND NOT #Stat_PosDesligando_Bool;   // rising edge of #Stat_AuxOutputLiga_Bool
   #Stat_PosDesligando_Bool := #Stat_AuxOutputLiga_Bool;
   IF #_w2 OR NOT #InOutCommand_Control.desligando THEN #Stat_AuxDesligando_Bool := FALSE; END_IF;
END_REGION

REGION Network 9: Falha Partida Não Desligou
   #Stat_FalhaDisjuntorNaoDesligou_TONTIME(IN := #InOutCommand_Control.desligando, PT := #inTempoFalha);   // TON
   IF #Stat_FalhaDisjuntorNaoDesligou_TONTIME.Q THEN
       #InOutCommand_Control.falhaPartidaNaoDesligou := TRUE;
   END_IF;
END_REGION

REGION Network 10: Falha Disjuntor Desligou
   #_w1 := NOT #inConfirmcaoDisjuntor AND #Stat_NegDisjuntor_Bool;   // falling edge of #inConfirmcaoDisjuntor
   #Stat_NegDisjuntor_Bool := #inConfirmcaoDisjuntor;
   IF #_w1 AND #InOutCommand_Control.ligado THEN #InOutCommand_Control.falhaDisjuntoDesligou := TRUE; END_IF;
END_REGION

REGION Network 11: Falha Confirmação Contator
   // Gera Falha Partida não confirmou
   #Stat_FalhaConfirmacao_TONTIME(IN := ((NOT #inConfirmacaoContator_Sentido1 AND NOT #Sentido_Giro) OR (NOT #inConfirmacaoContator_Sentido2 AND #Sentido_Giro)) AND #Stat_AuxOutputLiga_Bool,   // TON
                           PT := #inTempoFalha);
   IF #Stat_FalhaConfirmacao_TONTIME.Q THEN #InOutCommand_Control.falhaPartidaConfirmou := TRUE; END_IF;
END_REGION

REGION Network 12 (SCL): Falha Geral
       //Falha Geral
       IF #InOutCommand_Control.falhaPartidaConfirmou OR
           #InOutCommand_Control.falhaContatorDesligou OR
           #InOutCommand_Control.falhaDisjuntoDesligou OR
           #InOutCommand_Control.falhaPartidaNaoDesligou
       THEN
           #Static_Aux_Falha_Geral_Bool := true;
       ELSE
           #Static_Aux_Falha_Geral_Bool := false;
       END_IF;
END_REGION

REGION Network 13: Status Partida Ligada/Desligada
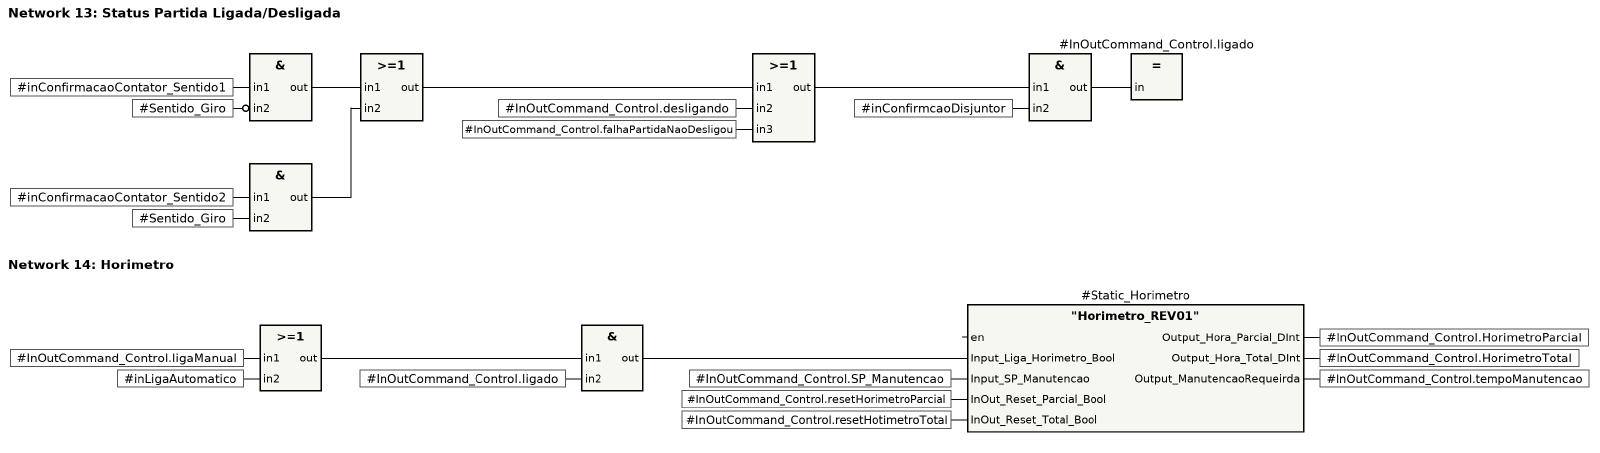
   #InOutCommand_Control.ligado := ((#inConfirmacaoContator_Sentido1 AND NOT #Sentido_Giro) OR (#inConfirmacaoContator_Sentido2 AND #Sentido_Giro) OR #InOutCommand_Control.desligando OR #InOutCommand_Control.falhaPartidaNaoDesligou) AND #inConfirmcaoDisjuntor;
END_REGION

REGION Network 14: Horimetro
   #Static_Horimetro(Input_Liga_Horimetro_Bool := (#InOutCommand_Control.ligaManual OR #inLigaAutomatico) AND #InOutCommand_Control.ligado,   // "Horimetro_REV01"
                     Input_SP_Manutencao := #InOutCommand_Control.SP_Manutencao,
                     InOut_Reset_Parcial_Bool := #InOutCommand_Control.resetHorimetroParcial,
                     InOut_Reset_Total_Bool := #InOutCommand_Control.resetHotimetroTotal,
                     Output_Hora_Parcial_DInt => #InOutCommand_Control.HorimetroParcial,
                     Output_Hora_Total_DInt => #InOutCommand_Control.HorimetroTotal,
                     Output_ManutencaoRequeirda => #InOutCommand_Control.tempoManutencao);
END_REGION

REGION Network 15 (SCL): Status Supervisorio
   //Sinais Supervisório
   #InOutCommand_Control.liberado := #Stat_Liberado_Motor;
   #InOutCommand_Control.emergencia := #inEmergencia;
   #InOutCommand_Control.disjuntorDesligado := NOT #inConfirmcaoDisjuntor;
END_REGION

REGION Network 16 (SCL): Reset Falhas
   //Reset Falhas
   IF #InOutCommand_Control.reset THEN

       #InOutCommand_Control.falhaPartidaConfirmou := false;
       #InOutCommand_Control.falhaContatorDesligou := false;
       #InOutCommand_Control.falhaDisjuntoDesligou := false;
       #InOutCommand_Control.falhaPartidaNaoDesligou := false;

       #InOutCommand_Control.reset := false;
   END_IF;
END_REGION
END_FUNCTION_BLOCK

FUNCTION_BLOCK "Atuador_Linear_Bifurcada"   // FB10, FBD
TITLE = Controle atuador com retorno de posição por fim de curso com dois lados (aberto, fechado)
{ S7_Optimized_Access := 'TRUE' }
VERSION : 0.1
// Maycon Lutz
// 15/07/20
// 
// Lado 1 - Considerado Aberto
// Lado 2 - Considerado Fechado
   VAR_INPUT
      inConfirmacao_Contator_Lado1 : Bool;
      inConfirmacao_Contator_Lado2 : Bool;
      inSensor_Lado1 : Bool;
      inSensor_Lado2 : Bool;
      inAciona_Lado1_Auto : Bool;
      inAciona_Lado2_Auto : Bool;
      inTempo_Falha : Time;
      inEmergencia : Bool;
      inLibera : Bool;
   END_VAR
   VAR_OUTPUT
      outAciona_Lado1 : Bool;
      outAciona_Lado2 : Bool;
      outEm_Posicao_Lado1 : Bool;
      outEm_Posicao_Lado2 : Bool;
   END_VAR
   VAR_IN_OUT
      Command : "typeAtuadorLinearDigital";
   END_VAR
   VAR
      Liberado : Bool;
      Intertravamento_Modo_Digital : Bool;
      Temporizador_Intertravamento : TON_TIME;
      Temporizador_Falha_Acionamento : TON_TIME;
      Temporizador_Falha_Contator_Lado1 : TON_TIME;
      Temporizador_Falha_Contator_Lado2 : TON_TIME;
      R_Trig_Manual : R_TRIG;
      R_Trig_Automatico : R_TRIG;
   END_VAR
BEGIN

REGION Network 1 (SCL): Controle modo Manual e Automático
   #R_Trig_Manual(CLK := #Command.Manual);
   //borda de subida em manual, false em automatico
   IF #R_Trig_Manual.Q THEN
       #Command.Automatico := false;
   END_IF;

   //borda de subida em automatico, false em manual
   #R_Trig_Automatico(CLK := #Command.Automatico);

   IF #R_Trig_Automatico.Q THEN
       #Command.Manual := false;
   END_IF;

   //Se os dois bits em true, false em automatico
   IF #Command.Manual AND #Command.Automatico THEN
       #Command.Automatico := false;
   END_IF;

   //se os dois bits em false, true em manual
   IF NOT #Command.Manual AND NOT #Command.Automatico THEN
       #Command.Manual := true;
   END_IF;
END_REGION

REGION Network 2 (SCL): Status Sensores
   #Command.Em_Posicao_Lado1 := #inSensor_Lado1;
   #Command.Em_Posicao_Lado2 := #inSensor_Lado2;
   #outEm_Posicao_Lado1 := #inSensor_Lado1;
   #outEm_Posicao_Lado2 := #inSensor_Lado2;
END_REGION

REGION Network 3 (SCL): Condições Liberação Funcionamento
   IF #inEmergencia AND //emergencia
       (#inLibera OR #Command.Libera_Bloqueio_Manual) AND //liberado
       NOT #Command.Falha_Acionando_Lado1 AND // falha acionamento lado 1
       NOT #Command.Falha_Acionando_Lado2 AND //falha acionamento lado 2
       NOT #Command.Falha_2_Posicoes_Ativa AND
       NOT #Command.Falha_Confirmacao_Contator_Lado1 AND
       NOT #Command.Falha_Confirmacao_Contator_Lado2 AND 
       NOT #Command.Manutencao AND // em manutenção
       NOT (#inAciona_Lado1_Auto AND #inAciona_Lado2_Auto)//acionado 2 lado ao mesmo tempo em auto
   THEN
       #Liberado := true;
   ELSE
       #Liberado := false;

       #Command.Aciona_Lado1 := false;
       #Command.Aciona_Lado2 := false;
   END_IF;
END_REGION

REGION Network 4 (SCL): Status das condições
   #Command.Em_Emergencia := #inEmergencia;
   #Command.Liberado := #Liberado;
END_REGION

REGION Network 5 (SCL): Acionamento

   IF #Command.Automatico THEN
       #Command.Aciona_Lado1 := false;
       #Command.Aciona_Lado2 := false;
   END_IF;



   //Verifica se estava acionado de um lado e foi solicitado outro lado
   //assim reseta o lado anterior e intertrava o lado novo solicitado
   //evitando problemas em campo.
   IF #Command.Aciona_Lado1 AND
       #Command.Aciona_Lado2 THEN

       #Intertravamento_Modo_Digital := true;

       IF #Command.Acionando_Lado1 THEN

           #Command.Aciona_Lado1 := false;
       END_IF;

       IF #Command.Acionando_Lado2 THEN

           #Command.Aciona_Lado2 := false;
       END_IF;

   END_IF;


   //temporizador de intertravamento quando solicitado dois lados ao mesmo tempo
   #Temporizador_Intertravamento(IN := #Intertravamento_Modo_Digital, PT := T#3S);

   //libera intertravamento
   IF #Temporizador_Intertravamento.Q THEN
       #Intertravamento_Modo_Digital := false;
   END_IF;


   //acionamento lado 1
   IF ((#Command.Aciona_Lado1 AND
       NOT #Intertravamento_Modo_Digital AND
       #Command.Manual) OR
       (#inAciona_Lado1_Auto AND
       #Command.Automatico
       ))
       AND #Liberado
   THEN

       //quando chegou na posição para de acionar e reseta o aciona lado
       IF #Command.Em_Posicao_Lado1 THEN
           #Command.Aciona_Lado1 := false;
           #Command.Acionando_Lado1 := false;
           #outAciona_Lado1 := false;

       ELSE
           //aciona lado 1
           #Command.Acionando_Lado1 := true;
           #outAciona_Lado1 := true;
       END_IF;
   ELSE

       #Command.Acionando_Lado1 := false;
       #outAciona_Lado1 := false;

   END_IF;

   //acionamento lado 2
   IF ((#Command.Aciona_Lado2 AND
       NOT #Intertravamento_Modo_Digital AND
       #Command.Manual) OR
       (#inAciona_Lado2_Auto AND
       #Command.Automatico
       ))
   //Não verifica se esta liberado ou não pois para fechar o registro não precisar estar liberado, somente para abrir.
   THEN

       //quando chegou na posição para de acionar e reseta o aciona lado
       IF #Command.Em_Posicao_Lado2 THEN
           #Command.Aciona_Lado2 := false;
           #Command.Acionando_Lado2 := false;
           #outAciona_Lado2 := false;
       ELSE
           //aciona lado 2
           #Command.Acionando_Lado2 := true;
           #outAciona_Lado2 := true;
       END_IF;
   ELSE

       #Command.Acionando_Lado2 := false;
       #outAciona_Lado2 := false;

   END_IF;
END_REGION

REGION Network 6 (SCL): Falha confirmação contatores

   #Temporizador_Falha_Contator_Lado1(IN := #outAciona_Lado1 AND NOT #inConfirmacao_Contator_Lado1,
                                      PT := t#3s);

   #Temporizador_Falha_Contator_Lado2(IN := #outAciona_Lado2 AND NOT #inConfirmacao_Contator_Lado2,
                                      PT := t#3s);

   IF #Temporizador_Falha_Contator_Lado1.Q THEN
       #Command.Falha_Confirmacao_Contator_Lado1 := true;
   END_IF;

   IF #Temporizador_Falha_Contator_Lado2.Q THEN
       #Command.Falha_Confirmacao_Contator_Lado2 := true;
   END_IF;
END_REGION

REGION Network 7 (SCL): Falha 2 posições ativas
   IF #Command.Em_Posicao_Lado1 AND #Command.Em_Posicao_Lado2 THEN
       #Command.Falha_2_Posicoes_Ativa := true;
   END_IF;
END_REGION

REGION Network 8 (SCL): Falha acionamento - Sensor não encontrado
   //conta tempo para falha de acionamento
   #Temporizador_Falha_Acionamento(IN := (#Command.Acionando_Lado1 OR #Command.Acionando_Lado2),
                                   PT := #inTempo_Falha);
   //falha de acionamento
   IF #Temporizador_Falha_Acionamento.Q THEN
       IF #Command.Acionando_Lado1 THEN
           #Command.Falha_Acionando_Lado1 := true;
       END_IF;

       IF #Command.Acionando_Lado2 THEN
           #Command.Falha_Acionando_Lado2 := true;
       END_IF;

   END_IF;
END_REGION

REGION Network 9 (SCL): Reset Falha
   //reset falha de acionamento
   IF #Command.Reset_Falha THEN
       #Command.Falha_Acionando_Lado1 := false;
       #Command.Falha_Acionando_Lado2 := false;
       #Command.Falha_2_Posicoes_Ativa := false;
       #Command.Falha_Confirmacao_Contator_Lado1 := false;
       #Command.Falha_Confirmacao_Contator_Lado2 := false;
       #Command.Reset_Falha := false;
   END_IF;
END_REGION
END_FUNCTION_BLOCK

FUNCTION_BLOCK "INV"   // FB14, FBD
{ S7_Optimized_Access := 'TRUE' }
VERSION : 0.1
   VAR_INPUT
      inHardwareID : Hw_Io;
      inEmergencia : Bool;
      inLibera : Bool;
      inLigaAutomatico : Bool;
      inVelocidadeAutomatica : Real;
      inRefSpeed : Real;
      inSimulacao : Bool;
   END_VAR
   VAR_OUTPUT
      outVelocidadeAtual : Real;
      outCorrente : Real;
      outPotencia : Real;
      outRampaAceleracao : Real;
      outRampaDesaceleracao : Real;
      outRotacaoMinima : Real;
      outRotacaoMaxima : Real;
      outCodigoAlarme : Real;
      outCodigoFalha : Real;
   END_VAR
   VAR_IN_OUT
      inOutControl : "typeINV";
   END_VAR
   VAR
      Static_SinaPara : "SINA_PARA";
      AxisEnabled : Bool;
      Lockout : Bool;
      Error : Bool;
      Status : Word;
      Diagld : Word;
      Static_SinaSpeed : "SINA_SPEED";
      Quantidade_Parametros : Int;   // Máximo 16 parametros Read/Write
      ConfigAxis : Word;
      Ready : Bool;
      Busy : Bool;
      Done : Bool;
      Error_1 : Bool;
      ErrorId : Real;
      Diagld_1 : Word;
      Velocidade_Desejada : Real;
      Horimetro : "Horimetro_REV01";
      Tempo_Limpeza : DInt;
      Stat_TOF_Desligamento : TOF_TIME;
   END_VAR
BEGIN

REGION Network 1: Parametros Read/Write
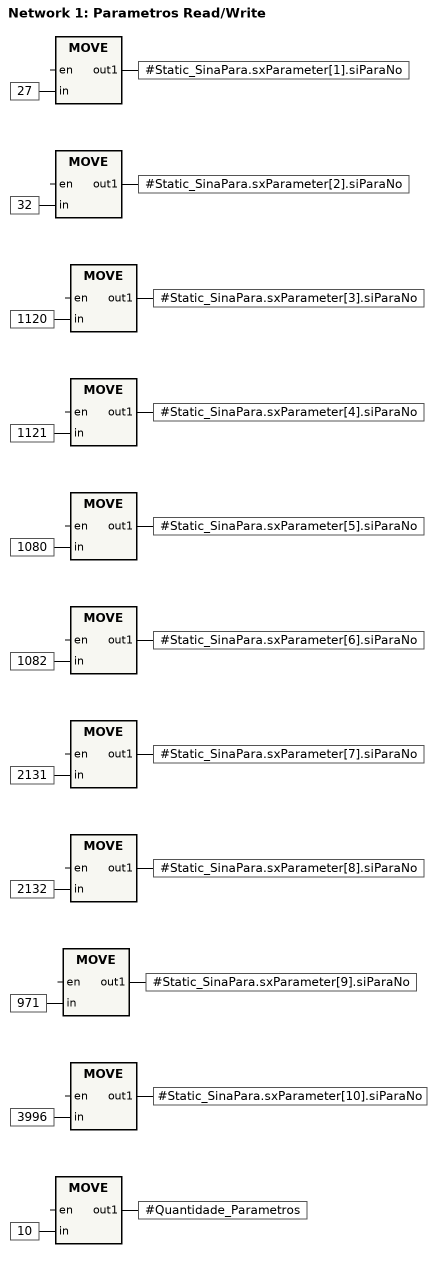
   #Static_SinaPara.sxParameter[1].siParaNo := 27;   // Corrente
   #Static_SinaPara.sxParameter[2].siParaNo := 32;   // Potência
   #Static_SinaPara.sxParameter[3].siParaNo := 1120;   // Rampa de Aceleração
   #Static_SinaPara.sxParameter[4].siParaNo := 1121;   // Rampa Desaceleração / Rampa de desacelração
   #Static_SinaPara.sxParameter[5].siParaNo := 1080;   // Rotação Minima / Rotação Mínima
   #Static_SinaPara.sxParameter[6].siParaNo := 1082;   // Rotação Máxima
   #Static_SinaPara.sxParameter[7].siParaNo := 2131;   // Código de Falha Atual / Código de Falha
   #Static_SinaPara.sxParameter[8].siParaNo := 2132;   // Código de Alarme Atual / Código de Alarme
   #Static_SinaPara.sxParameter[9].siParaNo := 971;   // Salva RAM TO ROM / Salva RAM to ROM
   #Static_SinaPara.sxParameter[10].siParaNo := 3996;   // r3996[0] - for diferente de 0, esta em progresso de escrita na ROM
   #Quantidade_Parametros := 10;
END_REGION

REGION Network 2: Leitura/ Escrita Parametros
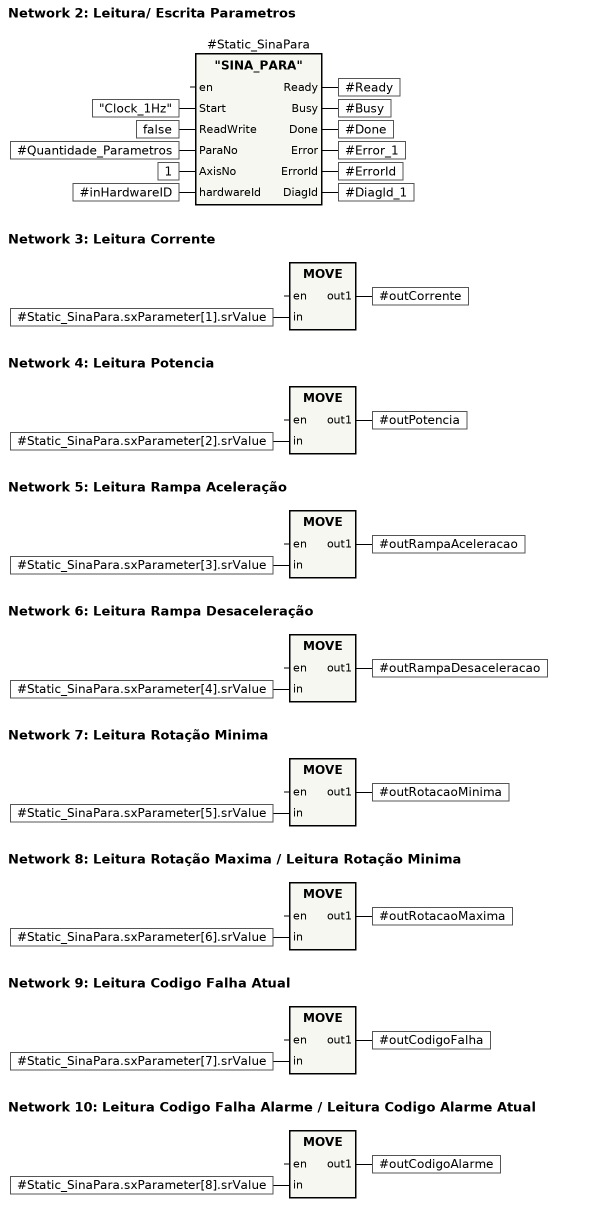
   #Static_SinaPara(Start := "Clock_1Hz",   // "SINA_PARA"
                    ReadWrite := false,
                    ParaNo := #Quantidade_Parametros,
                    AxisNo := 1,
                    hardwareId := #inHardwareID,
                    Ready => #Ready,
                    Busy => #Busy,
                    Done => #Done,
                    Error => #Error_1,
                    ErrorId => #ErrorId,
                    DiagId => #Diagld_1);
END_REGION

REGION Network 3: Leitura Corrente
   // Parametro: 27
   #outCorrente := #Static_SinaPara.sxParameter[1].srValue;
END_REGION

REGION Network 4: Leitura Potencia
   // Parametro: 32
   #outPotencia := #Static_SinaPara.sxParameter[2].srValue;
END_REGION

REGION Network 5: Leitura Rampa Aceleração
   // Parametro: 1120[0]
   #outRampaAceleracao := #Static_SinaPara.sxParameter[3].srValue;
END_REGION

REGION Network 6: Leitura Rampa Desaceleração
   // Parametro: 1121[0]
   #outRampaDesaceleracao := #Static_SinaPara.sxParameter[4].srValue;
END_REGION

REGION Network 7: Leitura Rotação Minima
   // Parametro: 1080
   #outRotacaoMinima := #Static_SinaPara.sxParameter[5].srValue;
END_REGION

REGION Network 8: Leitura Rotação Maxima / Leitura Rotação Minima
   // Parametro: 1082[0]
   #outRotacaoMaxima := #Static_SinaPara.sxParameter[6].srValue;
END_REGION

REGION Network 9: Leitura Codigo Falha Atual
   // Parametro: 2131
   #outCodigoFalha := #Static_SinaPara.sxParameter[7].srValue;
END_REGION

REGION Network 10: Leitura Codigo Falha Alarme / Leitura Codigo Alarme Atual
   // Parametro: 2132
   #outCodigoAlarme := #Static_SinaPara.sxParameter[8].srValue;
END_REGION

REGION Network 11: Assignment of the config Axis
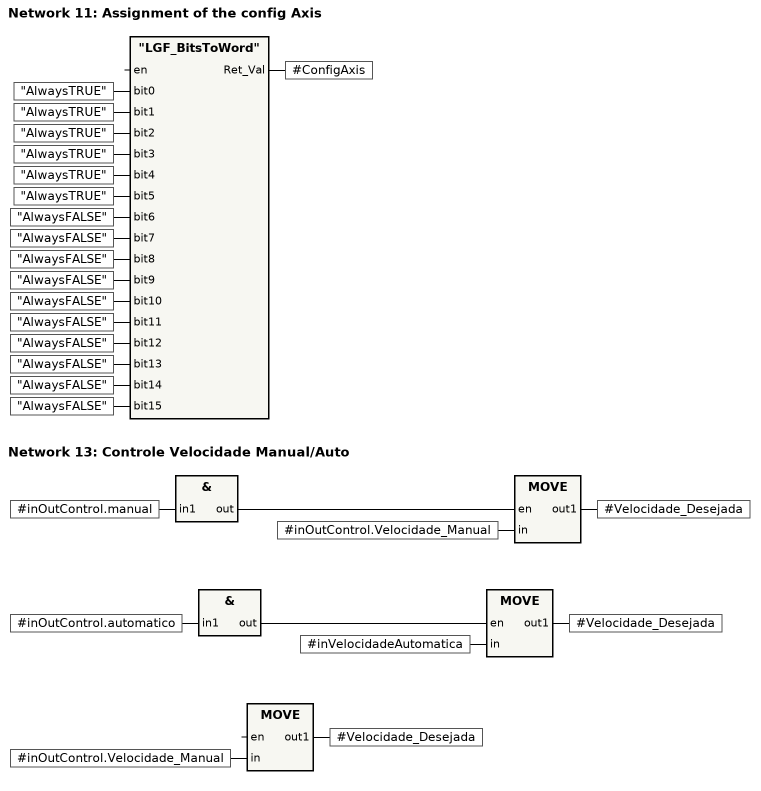
   #ConfigAxis := "LGF_BitsToWord"(bit0 := "AlwaysTRUE",
                           bit1 := "AlwaysTRUE",
                           bit2 := "AlwaysTRUE",
                           bit3 := "AlwaysTRUE",
                           bit4 := "AlwaysTRUE",
                           bit5 := "AlwaysTRUE",
                           bit6 := "AlwaysFALSE",
                           bit7 := "AlwaysFALSE",
                           bit8 := "AlwaysFALSE",
                           bit9 := "AlwaysFALSE",
                           bit10 := "AlwaysFALSE",
                           bit11 := "AlwaysFALSE",
                           bit12 := "AlwaysFALSE",
                           bit13 := "AlwaysFALSE",
                           bit14 := "AlwaysFALSE",
                           bit15 := "AlwaysFALSE");
END_REGION

REGION Network 12 (SCL): Controle modo Manual/Auto
   //Controle modos 
   IF NOT #inOutControl.manual AND NOT #inOutControl.automatico THEN
       #inOutControl.manual := true;
       //#InOutControl.Automatico := false;
   END_IF;

   IF #inOutControl.manual AND #inOutControl.automatico THEN
       #inOutControl.manual := true;
       //#InOutControl.Automatico := false;

   END_IF;
END_REGION

REGION Network 13: Controle Velocidade Manual/Auto
   IF #inOutControl.manual THEN #Velocidade_Desejada := #inOutControl.Velocidade_Manual; END_IF;
   IF #inOutControl.automatico THEN #Velocidade_Desejada := #inVelocidadeAutomatica; END_IF;
   #Velocidade_Desejada := #inOutControl.Velocidade_Manual;
END_REGION

REGION Network 14: Assignment of the config Axis
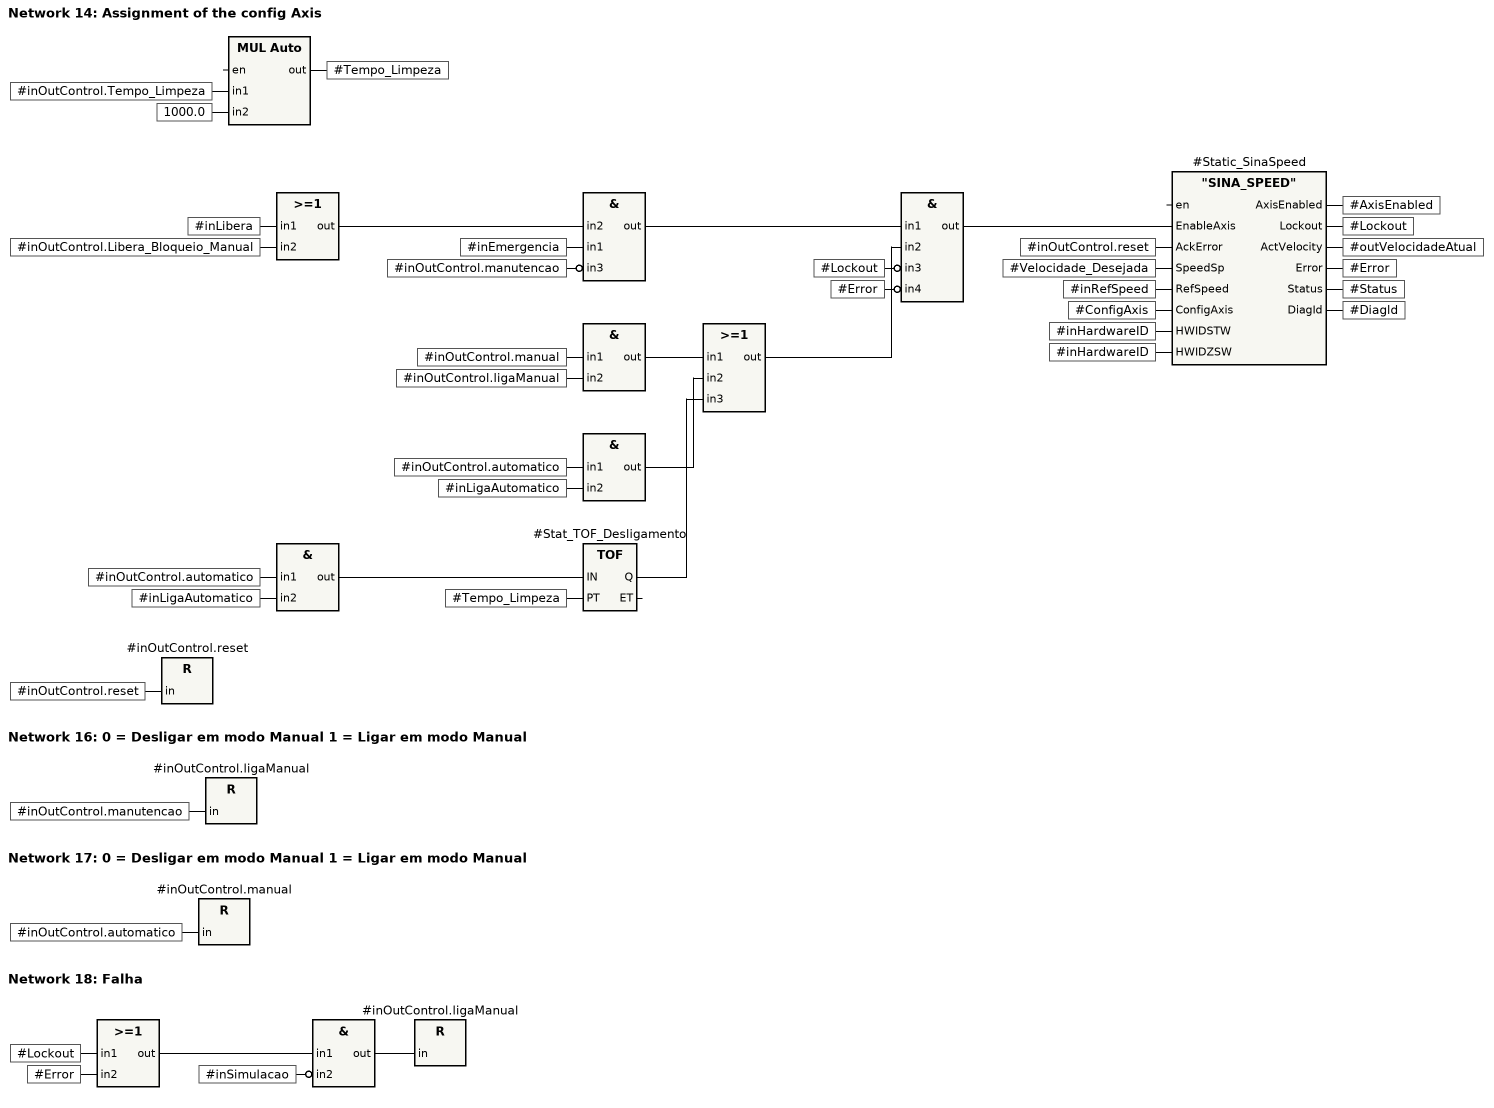
   #Tempo_Limpeza := #inOutControl.Tempo_Limpeza * 1000.0;
   #Stat_TOF_Desligamento(IN := #inOutControl.automatico AND #inLigaAutomatico, PT := #Tempo_Limpeza);   // TOF
   #Static_SinaSpeed(EnableAxis := (#inLibera OR #inOutControl.Libera_Bloqueio_Manual) AND #inEmergencia AND NOT #inOutControl.manutencao AND ((#inOutControl.manual AND #inOutControl.ligaManual) OR (#inOutControl.automatico AND #inLigaAutomatico) OR #Stat_TOF_Desligamento.Q) AND NOT #Lockout AND NOT #Error,   // "SINA_SPEED"
                     AckError := #inOutControl.reset,
                     SpeedSp := #Velocidade_Desejada,
                     RefSpeed := #inRefSpeed,
                     ConfigAxis := #ConfigAxis,
                     HWIDSTW := #inHardwareID,
                     HWIDZSW := #inHardwareID,
                     AxisEnabled => #AxisEnabled,
                     Lockout => #Lockout,
                     ActVelocity => #outVelocidadeAtual,
                     Error => #Error,
                     Status => #Status,
                     DiagId => #Diagld);
   IF #inOutControl.reset THEN #inOutControl.reset := FALSE; END_IF;
END_REGION

REGION Network 15 (SCL): Atualiza Palavra de comando
   IF NOT #inSimulacao THEN
       #inOutControl.Velocidade_Atual := #outVelocidadeAtual;
       #inOutControl.Corrente_Atual := #outCorrente;
       #inOutControl.Velocidade_Automatica_Solicitada := #inVelocidadeAutomatica;
       #inOutControl.Codigo_Falha := #outCodigoFalha;
       #inOutControl.Codigo_Alarme := #outCodigoAlarme;
   END_IF;
END_REGION

REGION Network 16: 0 = Desligar em modo Manual 1 = Ligar em modo Manual
   IF #inOutControl.manutencao THEN #inOutControl.ligaManual := FALSE; END_IF;
END_REGION

REGION Network 17: 0 = Desligar em modo Manual 1 = Ligar em modo Manual
   IF #inOutControl.automatico THEN #inOutControl.manual := FALSE; END_IF;
END_REGION

REGION Network 18: Falha
   IF (#Lockout OR #Error) AND NOT #inSimulacao THEN #inOutControl.ligaManual := FALSE; END_IF;
END_REGION

REGION Network 19: Status
   // 0 - Desligado
   // 1 - Ligado
   // 2 - Bloqueado
   // 3 - Em Modo Manutenção
   // 4 - Falha
   // 5 - Em Emergência
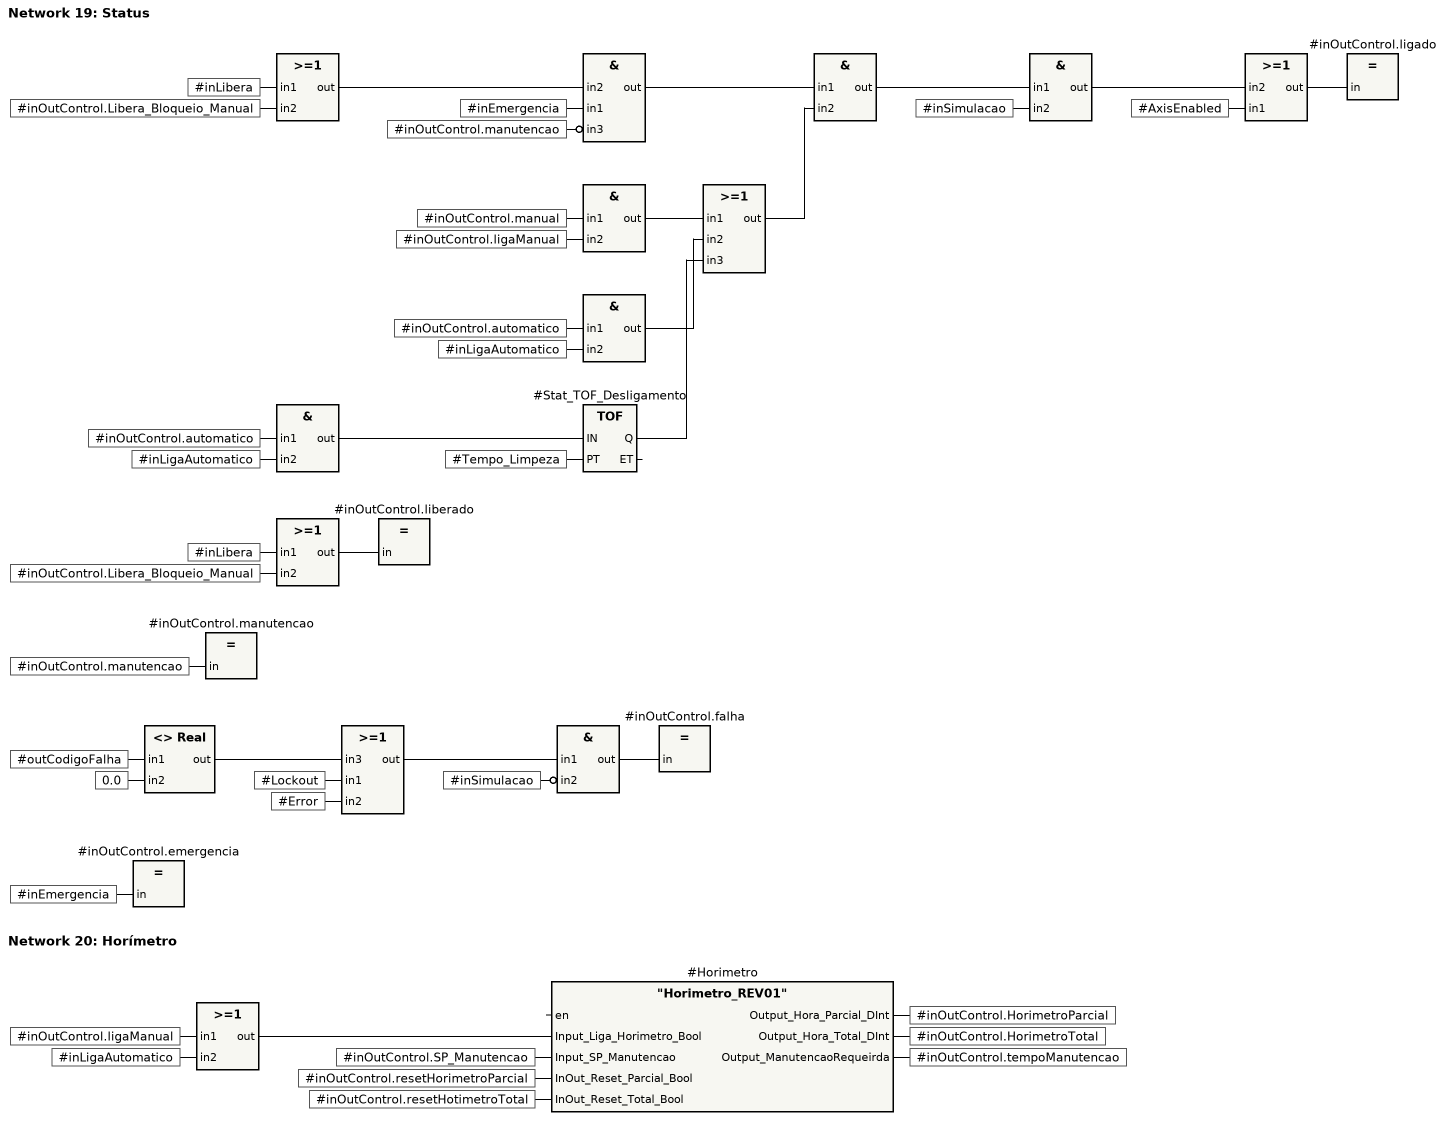
   #Stat_TOF_Desligamento(IN := #inOutControl.automatico AND #inLigaAutomatico, PT := #Tempo_Limpeza);   // TOF
   #inOutControl.ligado := ((#inLibera OR #inOutControl.Libera_Bloqueio_Manual) AND #inEmergencia AND NOT #inOutControl.manutencao AND ((#inOutControl.manual AND #inOutControl.ligaManual) OR (#inOutControl.automatico AND #inLigaAutomatico) OR #Stat_TOF_Desligamento.Q) AND #inSimulacao) OR #AxisEnabled;
   #inOutControl.liberado := #inLibera OR #inOutControl.Libera_Bloqueio_Manual;
   #inOutControl.manutencao := #inOutControl.manutencao;
   #inOutControl.falha := ((#outCodigoFalha <> 0.0) OR #Lockout OR #Error) AND NOT #inSimulacao;
   #inOutControl.emergencia := #inEmergencia;
END_REGION

REGION Network 20: Horímetro
   #Horimetro(Input_Liga_Horimetro_Bool := #inOutControl.ligaManual OR #inLigaAutomatico,   // "Horimetro_REV01"
              Input_SP_Manutencao := #inOutControl.SP_Manutencao,
              InOut_Reset_Parcial_Bool := #inOutControl.resetHorimetroParcial,
              InOut_Reset_Total_Bool := #inOutControl.resetHotimetroTotal,
              Output_Hora_Parcial_DInt => #inOutControl.HorimetroParcial,
              Output_Hora_Total_DInt => #inOutControl.HorimetroTotal,
              Output_ManutencaoRequeirda => #inOutControl.tempoManutencao);
END_REGION
END_FUNCTION_BLOCK

// folder: FC

FUNCTION "Read_Analogic_Wago" : Void   // FC2, SCL
{ S7_Optimized_Access := 'TRUE' }
VERSION : 0.1
   VAR_INPUT
      inValue : Int;
      inValueMax : Real;
   END_VAR
   VAR_OUTPUT
      outError : Bool;
      outValue : Real;
   END_VAR
BEGIN
   // <4.0mA  = 0x0003 - ERROR
   // 4mA     = 0x0000 - NO ERROR
   // 20mA    = 0x7FF8 - NO ERROR
   // >20.0mA = 0x7FFB - ERROR

   //Erro
   IF (#inValue.%X0 AND #inValue.%X1)
   THEN
       #outError := true;
   ELSE
       #outError := false;
   END_IF;

   IF #outError THEN

       #outValue := 0;
   ELSE
       #outValue := (#inValue/(32760/#inValueMax));
   END_IF;
END_FUNCTION

FUNCTION "Read_Analogic_Siemens" : Void   // FC3, SCL
{ S7_Optimized_Access := 'TRUE' }
VERSION : 0.1
   VAR_INPUT
      inValue : Int;
      inValueMax : Real;
   END_VAR
   VAR_OUTPUT
      outError : Bool;
      outValue : Real;
   END_VAR
BEGIN
   // <4.0mA  < 0  - ERROR
   // >20.0mA > 27648 - ERROR

   //Erro
   IF (#inValue > 27648) OR
       (#inValue < 0)
   THEN
       #outError := true;
   ELSE
       #outError := false;
   END_IF;

   IF #outError THEN

       #outValue := 0;
   ELSE
       #outValue := (#inValue/(27648/#inValueMax));
   END_IF;
END_FUNCTION